(*
触发缩回动作，成功触发返回TRUE，触发失败返回FALSE
*)
METHOD Act_DirectionJog : BOOL
VAR_IN_OUT
	_noteHMI:NoteStruct;
END_VAR
VAR_INPUT
	dir:BOOL;
	vel:DINT;
	len:DINT;
END_VAR
IF enable AND JOGCondition AND NOT busy THEN// AND NOT busy
	// pos:=0;
	// vel:=0;
	jogsetDir:=dir;
	jogsetlen:=len;
	IF (actpos-len>=minPos AND NOT dir) OR (actpos+len<=maxPos AND dir)THEN
		IF jogsetDir THEN
			FuncModule_RS232_ARM.ArmIN(pos:=actpos+len,vel:=setvel,acc:=10);
		ELSE
			FuncModule_RS232_ARM.ArmIN(pos:=actpos-len,vel:=setvel,acc:=10);
		END_IF
		note_IN:=FALSE;
		note_HOME:=FALSE;
		note_JOG:=FALSE;
		IF vel>0 THEN
			jogResetTime:=len/vel;
		END_IF
		jogBusy:=TRUE;
	ELSE
		note_IN:=FALSE;
		note_HOME:=FALSE;
		note_JOG:=TRUE;
		_noteHMI.showFlag:=TRUE;
		_noteHMI.showText:='';
		_noteHMI.showText:=CONCAT(_noteHMI.showText,nameTXT);
		_noteHMI.showText:=CONCAT(_noteHMI.showText,' JOG Condition Not Satisfied!');
	END_IF
	Act_DirectionJog:=TRUE;
ELSE
	Act_DirectionJog:=FALSE;
	note_IN:=FALSE;
	note_HOME:=FALSE;
	note_JOG:=TRUE;
	_noteHMI.showFlag:=TRUE;
	_noteHMI.showText:='';
	_noteHMI.showText:=CONCAT(_noteHMI.showText,nameTXT);
	_noteHMI.showText:=CONCAT(_noteHMI.showText,' JOG Condition Not Satisfied!');
END_IF
END_METHOD

(*
触发缩回动作，成功触发返回TRUE，触发失败返回FALSE
*)
METHOD Act_HOME : BOOL
VAR_IN_OUT
	_noteHMI:NoteStruct;
END_VAR
IF enable AND HOMECondition THEN// AND NOT busy
	// pos:=0;
	// vel:=0;
	Act_HOME:=HOME:=TRUE;
ELSE
	IF gCtrlMode=ControlMode.eManualCtrMode THEN
		note_IN:=FALSE;
		note_HOME:=FALSE;
		note_JOG:=TRUE;
		_noteHMI.showFlag:=TRUE;
		_noteHMI.showText:='';
		_noteHMI.showText:=CONCAT(_noteHMI.showText,nameTXT);
		_noteHMI.showText:=CONCAT(_noteHMI.showText,' HOME Condition Not Satisfied!');
	END_IF
	Act_HOME:=FALSE;
END_IF
END_METHOD

(*
触发缩回动作，成功触发返回TRUE，触发失败返回FALSE
*)
METHOD Act_HOME_Auto : BOOL
IF enable AND HOMECondition THEN// AND NOT busy
	// pos:=0;
	// vel:=0;
	Act_HOME_Auto:=HOME:=TRUE;
ELSE
	Act_HOME_Auto:=FALSE;
END_IF
END_METHOD

(*
触发伸出动作，成功触发返回TRUE，触发失败返回FALSE
*)
METHOD Act_IN : BOOL
VAR_IN_OUT
	_noteHMI:NoteStruct;
END_VAR
IF enable AND INCondition THEN// AND NOT busy
	// pos:=pos;
	// vel:=vel;
	Act_IN:=IN:=TRUE;
ELSE
	IF gCtrlMode=ControlMode.eManualCtrMode THEN
		note_IN:=TRUE;
		note_HOME:=FALSE;
		_noteHMI.showFlag:=TRUE;
		_noteHMI.showText:='';
		_noteHMI.showText:=CONCAT(_noteHMI.showText,nameTXT);
		_noteHMI.showText:=CONCAT(_noteHMI.showText,' IN Condition Not Satisfied!');
	END_IF
	Act_IN:=FALSE;
END_IF
END_METHOD

(*
触发伸出动作，成功触发返回TRUE，触发失败返回FALSE
*)
METHOD Act_IN_Auto : BOOL
IF enable AND INCondition THEN// AND NOT busy
	// pos:=pos;
	// vel:=vel;
	Act_IN_Auto:=IN:=TRUE;
ELSE
	Act_IN_Auto:=FALSE;
END_IF
END_METHOD

(*
触发复位报警动作，成功触发返回TRUE，触发失败返回FALSE
*)
METHOD Act_Reset : BOOL
VAR_INPUT
END_VAR
Act_Reset:=reset:=TRUE;
END_METHOD

(*
触发停止输出动作，成功触发返回TRUE，触发失败返回FALSE
*)
METHOD Act_Stop : BOOL
VAR_INPUT
END_VAR
Act_Stop:=stop:=TRUE;
END_METHOD

ACTION Error_ACT:
CASE errorStep OF
	0:
		error:=FALSE;
		errID:=0;
		errTXT:='';
 (*
	1:
		error:=TRUE;
		errID:=errorID+errorStep;
		errTXT:=CONCAT(STR1:=nameTXT,STR2:=' Extend Error!');
		errWTXT:=WCONCAT(STR1:=TO_WSTRING(nameTXT),STR2:=" 伸出(打开)错误");
	2:
		error:=TRUE;
		errID:=errorID+errorStep;
		errTXT:=CONCAT(STR1:=nameTXT,STR2:=' Retract Error!');
		errWTXT:=WCONCAT(STR1:=TO_WSTRING(nameTXT),STR2:=" 缩回(关闭)错误");
		*)
	1..5:
		error:=TRUE;
		errID:=getErrID(errorStep);
		errTXT:=getErrTXT(errorStep);
		errWTXT:=getErrWTXT(errorStep);
END_CASE
END_ACTION

METHOD Get_Done_HOME : BOOL
VAR_INPUT
END_VAR
Get_Done_HOME:=HOMEdone;
END_METHOD

METHOD Get_Done_IN : BOOL
VAR_INPUT
END_VAR
Get_Done_IN:=INdone;
END_METHOD

METHOD getErrID : UDINT
VAR_INPUT
	errID					:UDINT;//取值范围1~2
END_VAR
VAR
	nErrID					:UDINT;
END_VAR
nErrID:=errorID+errID;

getErrID:=nErrID;
END_METHOD

METHOD getErrTXT : STRING(255)
VAR_INPUT
	errID					:UDINT;//取值范围1~2
END_VAR
VAR
	sErrTXT					:STRING(255);
END_VAR

CASE errID OF
	1:
		sErrTXT:=CONCAT(STR1:=nameTXT,STR2:=' IN Error!');
	2:
		sErrTXT:=CONCAT(STR1:=nameTXT,STR2:=' HOME Error!');
	3:
		sErrTXT:=CONCAT(STR1:=nameTXT,STR2:=' SensorCheck Error!');
	4:
		sErrTXT:=CONCAT(STR1:=nameTXT,STR2:=' Home/IN Time Out Error!');
	5:
		sErrTXT:=CONCAT(STR1:=nameTXT,STR2:=' Communication Error!');
ELSE
	sErrTXT:=CONCAT(STR1:=nameTXT,STR2:='');
END_CASE
getErrTXT:=sErrTXT;
END_METHOD

METHOD getErrWTXT : WSTRING(255)
VAR_INPUT
	errID					:UDINT;//取值范围1~16
END_VAR
VAR
	sErrTXT					:WSTRING(255);
END_VAR

CASE errID OF
	1:
		sErrTXT:=WCONCAT(STR1:=TO_WSTRING(nameTXT),STR2:=" 去工作位错误");
	2:
		sErrTXT:=WCONCAT(STR1:=TO_WSTRING(nameTXT),STR2:=" 回原点错误");
	3:
		sErrTXT:=WCONCAT(STR1:=TO_WSTRING(nameTXT),STR2:=" 传感器检测异常");
	4:
		sErrTXT:=WCONCAT(STR1:=TO_WSTRING(nameTXT),STR2:=" 回原或去目标位超时异常");
	5:
		sErrTXT:=WCONCAT(STR1:=TO_WSTRING(nameTXT),STR2:=" 通讯异常");
ELSE
	sErrTXT:=WCONCAT(STR1:=TO_WSTRING(nameTXT),STR2:="");
END_CASE
getErrWTXT:=sErrTXT;
END_METHOD

ACTION HOME_ACT:
// ARMHOME--HOME 触发
IF HOME AND NOT HOMECondition THEN
	note_HOME:=TRUE;
	note_IN:=FALSE;
	note_JOG:=FALSE;
	NoteHMI.showFlag:=TRUE;
	NoteHMI.showText:='';
	NoteHMI.showText:=CONCAT(NoteHMI.showText,nameTXT);
	NoteHMI.showText:=CONCAT(NoteHMI.showText,' Home Condition Not Satisfied!');
	operatorLog.append(CONCAT(nameTXT,' HOME Not Done'));
END_IF
IF HOME AND enable AND HOMECondition THEN// AND NOT busy
	busy:=TRUE;
	IN:=FALSE;
	INdone:=FALSE;
	HOMEdone:=FALSE;
	INStep:=0;
	HOMEStep:=10;
	note_IN:=FALSE;
	note_HOME:=FALSE;
	note_JOG:=FALSE;
	readAndWriteLock:=TRUE;
	operatorLog.append(CONCAT(nameTXT,' HOME Done'));
	//errorStep:=0;
END_IF
HOME:=FALSE;
// Jog先不考虑，万不得已再使用
// IN ,Home,Jog任意一个Busy；则Recive程序先不动；分别进入程序没发送之类，之后一直采集位置，监控是否到位
CASE HOMEStep OF
0:
	//ready
	
10:
	HOMEErrorDelayTon(IN:=FALSE);
	HOMEDoneDelayTon(IN:=FALSE);
	HOMEStep:=20;
	INRelay:=FALSE;
	HOMERelay:=TRUE;
	FuncModule_RS232_ARM.readSopFlag:=FALSE;
	FuncModule_RS232_ARM.ArmHOME();
15:
	HomedelaycheckTON(IN:=TRUE,PT:=HomedelaycheckTime);
	IF HomedelaycheckTON.Q THEN
		HOMEStep:=20;
		HomedelaycheckTON(IN:=FALSE);
	END_IF
20:
	IF NOT HOMEAprSw OR HOMEAprSw THEN // 读取传感器状态  AND readPos=HomePos
		HOMEStep:=30;
		HOMEErrorDelayTon(IN:=FALSE);
		RETURN;
	END_IF
	HOMEErrorDelayTon(IN:=(NOT HOMEAprSw),PT:=errorDelayTime);// or readPos<>HomePos
	IF HOMEErrorDelayTon.Q THEN
		HOMEStep:=200;
		INdone:=FALSE;
		HOMEdone:=FALSE;
		errorStep:=4;
		HOMEErrorDelayTon(IN:=FALSE);
	END_IF
	
30:
	HOMEStep:=100;
	readAndWriteLock:=FALSE;
100:
	HOMEErrorDelayTon(IN:=(NOT HOMEAprSw),PT:=errorDelayTime);// rec pos=setpos or SW HOME Sensor
	IF HOMEErrorDelayTon.Q THEN
		//done:=FALSE;
		INdone:=FALSE;
		HOMEdone:=FALSE;
		errorStep:=2;
		HOMEStep:=200;
		RETURN;
	END_IF
	IF enableHOMEAprSw THEN
		HOMEDoneDelayTon(IN:=HOMEAprSw AND FuncModule_RS232_ARM.readSopFlag,PT:=doneDelayTimeShortHOME);
	ELSE
		HOMEDoneDelayTon(IN:=NOT enableHOMEAprSw,PT:=doneDelayTimeLongHOME);
	END_IF
	
	IF HOMEDoneDelayTon.Q THEN
		IF HOMEAprSw THEN
			busy:=FALSE;
			//done:=TRUE;
			INdone:=FALSE;
			HOMEdone:=TRUE;
			errorStep:=0;
			HOMEStep:=150;
		ELSE
			busy:=FALSE;
			//done:=TRUE;
			INdone:=FALSE;
			HOMEdone:=FALSE;
			errorStep:=2;
			HOMEStep:=200;
		END_IF
	END_IF
150:
	readAndWriteLock:=FALSE;
	HOMEStep:=0;
200:
	readAndWriteLock:=FALSE;
	HOMEStep:=0;
END_CASE
END_ACTION

ACTION IN_ACT:
//气缸伸出--IN 触发
IF IN AND NOT INCondition THEN
	note_IN:=TRUE;
	note_HOME:=FALSE;
	note_JOG:=FALSE;
	NoteHMI.showFlag:=TRUE;
	NoteHMI.showText:='';
	NoteHMI.showText:=CONCAT(NoteHMI.showText,nameTXT);
	NoteHMI.showText:=CONCAT(NoteHMI.showText,' IN Condition Not Satisfied!');
	operatorLog.append(CONCAT(nameTXT,' In Not Done'));
END_IF
IF IN AND enable AND INCondition THEN// AND NOT busy
	busy:=TRUE;
	HOME:=FALSE;
	INdone:=FALSE;
	HOMEdone:=FALSE;
	INStep:=10;
	HOMEStep:=0;
	note_IN:=FALSE;
	note_HOME:=FALSE;
	note_JOG:=FALSE;
	readAndWriteLock:=TRUE;
	operatorLog.append(CONCAT(CONCAT(nameTXT,' IN'),DINT_TO_STRING(setvel)));
	//errorStep:=0;
END_IF
IN:=FALSE;
// Jog先不考虑，万不得已再使用
// IN ,Home,Jog任意一个Busy；则Recive程序先不动；分别进入程序没发送之类，之后一直采集位置，监控是否到位
CASE INStep OF
0:
	//ready
	
10:
	INErrorDelayTon(IN:=FALSE);
	INDoneDelayTon(IN:=FALSE);
	IndelaycheckTON(IN:=FALSE);
	INStep:=15;
	INRelay:=TRUE;
	FuncModule_RS232_ARM.readSopFlag:=FALSE;
	FuncModule_RS232_ARM.ArmIN(pos:=setpos,vel:=setvel,acc:=10);
	// send:vel
	HOMERelay:=FALSE;
15:
	IndelaycheckTON(IN:=TRUE,PT:=IndelaycheckTime);
	IF IndelaycheckTON.Q THEN
		INStep:=20;
		IndelaycheckTON(IN:=FALSE);
	END_IF
20:
	IF NOT HOMEAprSw (*AND readPos=InPos*) THEN // 读取数据，判断接收的数据是否是设定的Vel；
		INStep:=30;
		INErrorDelayTon(IN:=FALSE);
		RETURN;
	ELSE
		INStep:=15;
	END_IF
	INErrorDelayTon(IN:=(HOMEAprSw (*OR readPos<>InPos*) ),PT:=errorDelayTime);
	IF INErrorDelayTon.Q THEN
		INStep:=200;
		INdone:=FALSE;
		HOMEdone:=FALSE;
		errorStep:=4;
		INErrorDelayTon(IN:=FALSE);
	END_IF
	
30:
	// send:pos
	INStep:=100;
	readAndWriteLock:=FALSE;
	
100:
	INErrorDelayTon(IN:=(HOMEAprSw OR NOT FuncModule_RS232_ARM.readSopFlag),PT:=errorDelayTime);// rec pos=setpos or SW IN Sensor
	IF INErrorDelayTon.Q THEN
		//done:=FALSE;
		INdone:=FALSE;
		HOMEdone:=FALSE;
		errorStep:=1;
		INStep:=200;
		RETURN;
	END_IF
	IF enableINAprSw THEN// Run则通过指令知道设备在什么地方
		INDoneDelayTon(IN:=NOT HOMEAprSw AND FuncModule_RS232_ARM.readSopFlag,PT:=doneDelayTimeShortIN);// rec pos=setpos
	ELSE
		INDoneDelayTon(IN:=NOT enableINAprSw,PT:=doneDelayTimeLongIN);
	END_IF
	
	IF INDoneDelayTon.Q THEN
		IF NOT HOMEAprSw THEN
			busy:=FALSE;
			//done:=TRUE;
			INdone:=TRUE;
			HOMEdone:=FALSE;
			errorStep:=0;
			INStep:=150;
		ELSE
			busy:=FALSE;
			//done:=TRUE;
			INdone:=FALSE;
			HOMEdone:=FALSE;
			errorStep:=1;
			INStep:=200;
		END_IF
	END_IF
150:
	readAndWriteLock:=FALSE;
	INStep:=0;
200:
	readAndWriteLock:=FALSE;
	INStep:=0;
END_CASE
END_ACTION

ACTION Init_ACT:
done:=(INdone OR HOMEdone);
InitHMI_ACT();
manualCtrl_ACT();

IF NOT FuncModule_RS232_ARM.serialConnected AND firstPowerTON.Q THEN
	errorStep:=5;
END_IF
noteTON_P(IN:=note_IN,PT:=T#0.1S);
noteRTrig_P(CLK:=noteTON_P.Q);
IF noteRTrig_P.Q THEN
//	gLog_Note.append_EX(noteWTXT_Ext);
END_IF
noteTON_N(IN:=note_HOME,PT:=T#0.1S);
noteRTrig_N(CLK:=noteTON_N.Q);
IF noteRTrig_N.Q THEN
//	gLog_Note.append_EX(noteWTXT_Ret);
END_IF

jogResetTON(in:=jogBusy,PT:=DINT_TO_TIME(jogResetTime*1000));
IF jogResetTON.Q THEN
	jogBusy:=FALSE;
END_IF
END_ACTION

ACTION InitHMI_ACT:
HMIItf.INAprSw:=INAprSw;
HMIItf.HOMEAprSw:=HOMEAprSw;
HMIItf.enableIN:=enableINAprSw;
HMIItf.enableHOME:=enableHOMEAprSw;
HMIItf.HMIEnable:=hmiEN;
HMIItf.enable:=enable;
HMIItf.done:=done;
HMIItf.busy:=busy;
HMIItf.error:=error;
HMIItf.errID:=UDINT_TO_DINT(errID);
HMIItf.errTXT:=errTXT;
HMIItf.INRelay:=INRelay;
HMIItf.HOMERelay:=HOMERelay;
HMIItf.power:=power;
HMIItf.nameTXT:=nameTXT;
HMIItf.extenderror:=error AND errorID=1;
HMIItf.retracterror:=error AND errorID=2;
HMIItf.INcondition:=INCondition;
HMIItf.HOMEcondition:=HOMECondition;
END_ACTION

ACTION ManualCtrl_ACT:
//HMI手动控制
//IF ctrlMode=eManualCtrMode THEN
IF hmiEN THEN
	INTrigRAlc(CLK:=HMIItf.INAndHOME);
	IF INTrigRAlc.Q THEN// AND NOT busy
		IF INRelay THEN//如果伸出继电器或伸出传感器亮，则认为已经伸出过
			HOME:=TRUE;
		END_IF
		IF HOMERelay THEN
			IN:=TRUE;
		END_IF
		IF NOT INRelay AND NOT HOMERelay THEN
			IF INAprSw THEN
				HOME:=TRUE;
			END_IF
			IF HOMEAprSw THEN
				IN:=TRUE;
			END_IF
		END_IF
	END_IF
	INTrigR1(CLK:=HMIItf.IN);
	IF INTrigR1.Q THEN// AND NOT busy
		WarmHMI.showText:='';
		WarmHMI.showFlag:=TRUE;
		WarmHMI.showText:=CONCAT(WarmHMI.showText,'Are you sure you want the ');
		WarmHMI.showText:=CONCAT(WarmHMI.showText,nameTXT);
		WarmHMI.showText:=CONCAT(WarmHMI.showText,' to INChamber?');
	END_IF
	IF WarmHMI.bOK AND NOT WarmHMI.showFlag AND FIND(WarmHMI.showText,nameTXT)>0 AND FIND(WarmHMI.showText,'INChamber')>0 THEN
		IN:=TRUE;
		WarmHMI.bOK:=FALSE;
		WarmHMI.showText:='';
	END_IF
	IF WarmHMI.bNO AND NOT WarmHMI.showFlag AND FIND(WarmHMI.showText,nameTXT)>0 AND FIND(WarmHMI.showText,'INChamber')>0 THEN
		WarmHMI.bNO:=FALSE;
		WarmHMI.showText:='';
	END_IF
	
	HOMETrigR1(CLK:=HMIItf.HOME);
	IF HOMETrigR1.Q THEN// AND NOT busy
		WarmHMI.showText:='';
		WarmHMI.showFlag:=TRUE;
		WarmHMI.showText:=CONCAT(WarmHMI.showText,'Are you sure you want to the ');
		WarmHMI.showText:=CONCAT(WarmHMI.showText,nameTXT);
		WarmHMI.showText:=CONCAT(WarmHMI.showText,' to Homing?');
	END_IF
	IF WarmHMI.bOK AND NOT WarmHMI.showFlag AND FIND(WarmHMI.showText,nameTXT)>0 AND FIND(WarmHMI.showText,'Homing')>0 THEN
		HOME:=TRUE;
		WarmHMI.bOK:=FALSE;
		WarmHMI.showText:='';
	END_IF
	IF WarmHMI.bNO AND NOT WarmHMI.showFlag AND FIND(WarmHMI.showText,nameTXT)>0 AND FIND(WarmHMI.showText,'Homing')>0 THEN
		WarmHMI.bNO:=FALSE;
		WarmHMI.showText:='';
	END_IF
	
	resetTrigR1(CLK:=HMIItf.reset);
	IF resetTrigR1.Q THEN// AND NOT busy
		reset:=TRUE;
	END_IF
	
	stopTrigR1(CLK:=HMIItf.stop);
	IF stopTrigR1.Q THEN// AND NOT busy
		stop:=TRUE;
	END_IF
	
	powerTrigR1(CLK:=HMIItf.power);
	IF powerTrigR1.Q THEN// AND NOT busy
		IF power THEN
			power:=FALSE;
		ELSE
			power:=TRUE;
		END_IF
	END_IF
END_IF
END_ACTION

ACTION Read_ACT:
//气缸收回--read 触发
firstPowerTON(IN:=firstPower,PT:=T#5S);
IF NOT readAndWriteLock AND NOT readbusy AND readStep=0 AND readCondition THEN// AND NOT busy
	readdone:=FALSE;
	readStep:=10;
	readbusy:=TRUE;
	readerror:=FALSE;
END_IF
CASE readStep OF
0:
	//ready
	readTon1(IN:=FALSE);
	readTon2(IN:=FALSE);
10:// State
	IF readAndWriteLock THEN
		readStep:=5000;
	ELSE
		FuncModule_RS232_ARM.readPosFlag:=FALSE;
		FuncModule_RS232_ARM.GetPos();
		readStep:=readStep+10;
	END_IF
20:
	IF readAndWriteLock THEN
		readStep:=5000;
	ELSE
		IF FuncModule_RS232_ARM.readPosFlag THEN
			FuncModule_RS232_ARM.readPosFlag:=FALSE;
			// 数据处理
			actpos:=FuncModule_RS232_ARM.POS;
			readTon1(IN:=FALSE);
			readStep:=25;
			RETURN;
		END_IF
		readTon1(IN:=TRUE,PT:=T#500MS);// 超时
		IF readTon1.Q THEN
			readStep:=6000;
			readTon1(IN:=FALSE);
			readTon2(IN:=FALSE);
			RETURN;
		END_IF
		;
	END_IF
25:
	t1(IN:=TRUE,PT:=T#0.5S);
	IF t1.Q THEN
		readStep:=5000;
		t1(IN:=FALSE);
	END_IF
100:// Internal RTD1
	IF readAndWriteLock THEN
		readStep:=5000;
	ELSE
		FuncModule_RS232_ARM.readStateFlag:=FALSE;
		FuncModule_RS232_ARM.GetState();
		readStep:=readStep+10;
	END_IF	
110:
	IF readAndWriteLock THEN
		readStep:=5000;
	ELSE
		IF FuncModule_RS232_ARM.readStateFlag THEN
			FuncModule_RS232_ARM.readStateFlag:=FALSE;
			// 数据处理
			readTon1(IN:=FALSE);
			readStep:=5000;
			RETURN;
		END_IF
		readTon1(IN:=TRUE,PT:=T#500MS);// 超时
		IF readTon1.Q THEN
			readStep:=6000;
			readTon1(IN:=FALSE);
			readTon2(IN:=FALSE);
			RETURN;
		END_IF
		;
	END_IF
	
5000:
	readbusy:=FALSE;
	readdone:=TRUE;
	readStep:=0;
	readerror:=FALSE;
6000:
	readbusy:=FALSE;
	readdone:=TRUE;
	readStep:=0;
	readerror:=TRUE;
END_CASE
END_ACTION

ACTION RealMonitor_ACT:
notBusyMonitorDelayTon(IN:=NOT busy,PT:=notBusyMonitorDelayTime);
IF real_TimeMonitor THEN
	IF notBusyMonitorDelayTon.Q THEN
		//伸出实时检测
//		IF (enableINAprSw AND NOT INAprSw) AND INRelay THEN
//			errorStep:=1;
//		END_IF
	
//		//缩回实时检测	
//		IF (enableINAprSw AND NOT HOMEAprSw) AND HOMERelay  THEN
//			errorStep:=2;
//		END_IF
	END_IF
END_IF
END_ACTION

ACTION Reset_ACT:
IF reset THEN
	IF NOT power THEN
		INRelay:=FALSE;
		HOMERelay:=FALSE;
	END_IF
	busy:=FALSE;
	//done:=FALSE;
	//extdone:=FALSE;
	//retdone:=FALSE;
	errorStep:=0;
	note_IN:=FALSE;
	note_HOME:=FALSE;
	note_JOG:=FALSE;
	reset:=FALSE;
END_IF

IF stop THEN
	stop:=FALSE;
	INRelay:=FALSE;
	HOMERelay:=FALSE;
	note_IN:=FALSE;
	note_HOME:=FALSE;
	note_JOG:=FALSE;
	busy:=FALSE;
	INStep:=0;
	HOMEStep:=0;
	FuncModule_RS232_ARM.ArmStop();
	//无自锁检测说法，直接停
//	extStep:=0;
//	retStep:=0;
END_IF
END_ACTION

ACTION VersionLog:
(*
版本: V1.0.0.0
说明:
	1. 首个版本
	2. 含普通气缸\真空吸类型的控制
	3. 可配置是否有到位信号, 以及到位稳定时间
(--------------------------------------------------)
新版本: V1.0.1.0
更新时间: 2019/11/20 19:00
更新说明:
	1. 优化编写方式
	2. 修改错误编码起始位，现改为从1开始
(--------------------------------------------------)
新版本: V1.0.1.1
更新时间: 2020/03/23 23:00
更新说明:
	1. 优化报错方式
	2. 增加伸出、缩回、复位和停止触发函数
(--------------------------------------------------)
新版本: V1.0.1.2
更新时间: 2020/04/22 09:50
更新说明:
	1. 增加中文报警输出
(--------------------------------------------------)
新版本: V1.0.1.3
更新时间: 2020/09/16
更新说明:
	1. 开放错误ID、错误文本信息获取接口
(--------------------------------------------------)
新版本: V1.0.1.4
更新时间: 2020/10/06
更新说明:
	1. 移除控制模式变量，增加HMI启用条件
	2. 增加外部获取伸出缩回完成信号接口函数
(--------------------------------------------------)
新版本: V1.0.1.5
更新时间: 2020/10/14
更新说明:
	1. 优化代码
(--------------------------------------------------)
*)
END_ACTION

END_FUNCTION_BLOCK

// ---- POUs/BaseModule/Communication/FuncModule_RS232_ARM.TcPOU
PROGRAM FuncModule_RS232_ARM
VAR_INPUT
	serialExcute				:BOOL;// RS232开始一次参数读取
	serialSlaveID				:UINT;// 232从站节点号
	sendstr						:STRING;
	prefix						:STRING:='';// 字符串头
	suffix						:STRING:= '';// 字符串尾
	timeout						:TIME:=T#200MS;// 超时时间
	goPosLoad					:LREAL;
	goPosPhase					:LREAL;
	setPresetExt				:BOOL;
	readPosFlag					:BOOL;
	readStateFlag				:BOOL;
	readSopFlag					:BOOL;// 停止标志位
END_VAR
VAR_OUTPUT
	serialBusy						:BOOL;
	setPresetBusy					:BOOL;
	serialDone						:BOOL;
	setPresetDone						:BOOL;
	serialError						:BOOL;
	setPresetError						:BOOL;
	serialConnected					:BOOL;
	POS							:INT;// 
	oldPOS							:int;// 
	phase							:REAL;// Phase电容
	rec_ManulOrAuto					:BOOL;// Manul OR Auto
	rec_MAStr						:STRING:='Auto';
	loadRunErr						:BOOL;
	phashRunErr						:BOOL;
END_VAR
VAR
	//Byte方式
	send1:							SendData;
	receive1:						ReceiveString;
 
	Timer1:							TON;
	TimerSetPreset:							TON;
	t1:								TON;
	ITemp:INT;
	arr_SendData:					STRING;(*READ*)//发送数据
	arr_RcvDataString:				STRING;// 接收数据
	arr_RcvDataStringTemp:				STRING;// 接收数据
	arr_RcvDataStringClear:			STRING;// 清除接收数据
	RcvDataFlag:			BOOL;// 接收数据标志位
	serialStep						:UINT;				//处理步数
	serialErrorID					:UINT;
	setPresetStep					:UINT;				//处理步数
	serialTimeOut:BOOL;//接收数据超时
	serialRecError:BOOL;//接收数据错误
	reciveFtrig:F_TRIG;
	recTon:TON;
	againSendS3:TON;
	//字符串方式
	(*send1:							SendString;
	receive1:						ReceiveString;
	
	Timer1:							TON;
	
	_sendString:					STRING:='4567';
	_receive1string:				STRING;
	_recvLast:						STRING;				//保存上一个周期接收的字符*)

	
	decimalvalue:INT;
	decimalvalueP:INT;
	hexString:STRING(8);
	hexStringP:STRING(8);
	i:INT;
	hexChars:ARRAY [0..15] OF STRING[1]:=['0','1','2','3','4','5','6','7','8','9','A','B','C','D','E','F'];
	index:INT;
	findposstart	:INT;
	findposend		:INT;
	find_pos		:INT;
	recStrTemp		:STRING(255);
END_VAR

(*
 *功能块的作用，把 TxBuffer 缓存区的数据经过 Process Data 的 ComOut 发送出去，
 *而把 ComIn 中的数据接收到 RxBuffer。引用这个功能块的程序执行周期越短，
 *数据交换的效率就越高，所以这段程序应该放在快速任务中作为 Backgroud 代码无条件执行。
*)
IF receive1.Error <> COMERROR_NOERROR THEN
	serialRecError:=TRUE;
END_IF
receive1(
	Prefix:= prefix, 
	Suffix:= suffix, 
	Timeout:=timeout , 
	Reset:= , 
	StringReceived=> , 
	Busy=> , 
	Error=> , 
	RxTimeout=> , 
	ReceivedString:= arr_RcvDataStringTemp, 
	RXbuffer:=gRxBuffer_ARM );

//testReal:=BYTE_TO_REAL(arr_RcvData_Temp);
//数据接收处理
reciveFtrig(CLK:=receive1.busy);
IF reciveFtrig.Q THEN
	arr_RcvDataString:=arr_RcvDataStringTemp;
	arr_RcvDataStringTemp:=arr_RcvDataStringClear;
	RcvDataFlag:=TRUE;
	serialConnected:=TRUE;
END_IF
recTon(IN:=RcvDataFlag, PT:=T#20MS);
IF recTon.Q THEN
	RcvDataFlag:=FALSE;
END_IF
againSendS3(IN:=NOT RcvDataFlag,PT:=T#5S);
IF againSendS3.Q THEN
	serialConnected:=FALSE;
	againSendS3(IN:=FALSE);
END_IF

ACT_Send();

ACT_RcvProcess();

ACTION ACT_RcvProcess:
find_pos:=0;
findposend:=0;
findposstart:=0;

IF MID(arr_RcvDataString,3,1)='?96' THEN
	recStrTemp:=DELETE(arr_RcvDataString,5,1);
	IF MID(recStrTemp,5,1)='Px.1='  THEN
		readPosFlag:=TRUE;
		IF  MID(recStrTemp,1,6)='-' THEN
			POS:=oldPOS+STRING_TO_INT(MID(recStrTemp,LEN(recStrTemp)-7,6));
		ELSE
			POS:=STRING_TO_INT(MID(recStrTemp,LEN(recStrTemp)-7,6));
			oldPOS:=POS;
		END_IF
	END_IF
END_IF

IF FIND(arr_RcvDataString,'Ux.1=8')>0 THEN
	readSopFlag:=TRUE;
END_IF
END_ACTION

ACTION ACT_Send:

CASE serialStep OF
	0:
	IF serialExcute THEN
		serialExcute:=FALSE;
		IF NOT serialBusy THEN
			serialStep:=90;
			serialBusy:=TRUE;
			serialDone:=FALSE;
			serialError:=FALSE;
			serialTimeOut:=FALSE;
			serialRecError:=FALSE;
		END_IF
	END_IF
	Timer1(IN:= FALSE);
	;
	90:
		arr_SendData:=sendstr;
		serialStep:=100;
	100:
		send1(
			pSendData:= ADR(arr_SendData), 
			Length:= INT_TO_UDINT(LEN(arr_SendData)), 
			Busy=> , 
			Error=> , 
			TXbuffer:= gTxBuffer_ARM);
		serialStep:=serialStep+10;
	110:
		Timer1(IN:= NOT timer1.q, PT:=T#10MS);
		IF Timer1.Q THEN
			serialStep:=serialStep+10;
			Timer1(IN:= FALSE);
		END_IF
	120:
		Timer1(IN:= NOT timer1.q, PT:=T#500MS);
		IF Timer1.Q THEN
			serialStep:=6000;
			Timer1(IN:= FALSE);
			serialTimeOut:=TRUE;
			RETURN;
		END_IF
		IF NOT send1.busy  THEN
			Timer1(IN:= FALSE);
			serialTimeOut:=FALSE;
			serialStep:=200;
		END_IF
		IF send1.Error <> COMERROR_NOERROR THEN
			serialRecError:=TRUE;
		END_IF
	200://数据处理
		serialStep:=serialStep+10;
	210:
		Timer1(IN:= NOT timer1.q, PT:=T#10MS);
		IF Timer1.Q THEN
			serialStep:=serialStep+10;
			Timer1(IN:= FALSE);
		END_IF
	220:
		//数据转换
		Timer1(IN:= FALSE);
		serialStep:=1000;
	
	1000:
		Timer1(IN:= NOT timer1.q, PT:=T#50MS);
		IF Timer1.Q THEN
			serialStep:=5000;
			Timer1(IN:= FALSE);
			// sendstr:='';
			serialTimeOut:=FALSE;
		END_IF
	;
	5000://done
		serialBusy:=FALSE;
		serialDone:=TRUE;
		serialError:=FALSE;
		serialStep:=0;
	;
	6000://error
		serialBusy:=FALSE;
		serialDone:=FALSE;
		serialError:=TRUE;
		serialStep:=0;
	;
	
END_CASE
END_ACTION

METHOD ArmHOME : BOOL
VAR_INPUT
END_VAR
sendstr:='';
sendstr:='|$R';
serialExcute:=TRUE;
END_METHOD

METHOD ArmIN : BOOL
VAR_INPUT
	pos:DINT;
	vel:DINT;
	acc:DINT;
END_VAR
VAR
	str:STRING;
END_VAR
str:='';
str:=CONCAT(str,'P=');
str:=CONCAT(str,DINT_TO_STRING(pos));
str:=CONCAT(str,',S=');
str:=CONCAT(str,DINT_TO_STRING(vel));
str:=CONCAT(str,',A=');
str:=CONCAT(str,DINT_TO_STRING(acc));
str:=CONCAT(str,',^$R');
sendstr:='';
sendstr:=str;
serialExcute:=TRUE;
END_METHOD

METHOD ArmStop : BOOL
VAR_INPUT
END_VAR
VAR
	diraction:STRING:='+';
	str:STRING;
END_VAR
str:='';
str:=CONCAT(str,']$R');
sendstr:='';
sendstr:=str;
serialExcute:=TRUE;
END_METHOD

METHOD CalASII_Str : STRING
VAR_INPUT
	date1:UINT;
END_VAR
IF date1=10 THEN
	CalASII_Str:='A';
END_IF
IF date1=11 THEN
	CalASII_Str:='B';
END_IF
IF date1=12 THEN
	CalASII_Str:='C';
END_IF
IF date1=13 THEN
	CalASII_Str:='D';
END_IF
IF date1=14 THEN
	CalASII_Str:='E';
END_IF
IF date1=15 THEN
	CalASII_Str:='F';
END_IF
IF date1<10 THEN
	CalASII_Str:=UINT_TO_STRING(date1);
END_IF
IF date1>15 THEN
	CalASII_Str:=UINT_TO_STRING(date1);
END_IF
END_METHOD

METHOD CalMeth : INT
VAR_INPUT
	byteIn:BYTE;
END_VAR
VAR_OUTPUT
	outInt:INT;
END_VAR
IF byteIn>=48 AND byteIn<=57 THEN
	outInt:=byteIn-48;
ELSE
	outInt:=byteIn-65+10;
END_IF
CalMeth:=outInt;
END_METHOD

METHOD GetPos : BOOL
VAR_INPUT
END_VAR
VAR
	str:STRING;
END_VAR
str:='?96$R';
sendstr:='';
sendstr:=str;
serialExcute:=TRUE;
END_METHOD

METHOD GetState : BOOL
VAR_INPUT
END_VAR
VAR
	str:STRING;
END_VAR
str:='GetState^';
sendstr:='';
sendstr:=str;
serialExcute:=TRUE;
END_METHOD

METHOD IncN : BOOL
VAR_INPUT
	dis:DINT;
	vel:DINT;
	acc:DINT;
END_VAR
VAR
	diraction:STRING:='+';
	str:STRING;
END_VAR
str:='';
str:=CONCAT(str,'P:');
str:=CONCAT(str,DINT_TO_STRING(dis));
str:=CONCAT(str,',S:');
str:=CONCAT(str,DINT_TO_STRING(vel));
str:=CONCAT(str,',A:');
str:=CONCAT(str,DINT_TO_STRING(acc));
str:=CONCAT(str,',D:');
str:=CONCAT(str,diraction);
str:=CONCAT(str,',^$R');
sendstr:='';
sendstr:=str;
serialExcute:=TRUE;
END_METHOD

METHOD IncP : BOOL
VAR_INPUT
	dis:DINT;
	vel:DINT;
	acc:DINT;
END_VAR
VAR
	diraction:STRING:='+';
	str:STRING;
END_VAR
str:='';
str:=CONCAT(str,'P:');
str:=CONCAT(str,DINT_TO_STRING(dis));
str:=CONCAT(str,',S:');
str:=CONCAT(str,DINT_TO_STRING(vel));
str:=CONCAT(str,',A:');
str:=CONCAT(str,DINT_TO_STRING(acc));
str:=CONCAT(str,',D:');
str:=CONCAT(str,diraction);
str:=CONCAT(str,',^$R');
sendstr:='';
sendstr:=str;
serialExcute:=TRUE;
END_METHOD

END_PROGRAM

// ---- POUs/BaseModule/ActionModule/RFModule_Source/RFModule_Source.TcPOU
(*
--报错编号0: 无报错
--报错编号1: openend Error
--报错编号2: close Error
*)
FUNCTION_BLOCK RFModule_Source
VAR_IN_OUT
	WarmHMI					:WARMStruct;
	NoteHMI					:NoteStruct;
	operatorLog				:printLogModule_EX;
END_VAR
VAR_INPUT
	HMIItf						:RFHMIStruts;// 每个RF对象都关联了一个HMI
	RFTYPE						:RFType:=RFType_Default;// 设置RF的类型
	real_TimeMonitor			:BOOL:=TRUE;//实时状态检测
	co_control					:BOOL;// 共同计时
	open						:BOOL:=FALSE;//启动触发信号
	openCondition				:BOOL:=TRUE;//启动条件
	close						:BOOL:=FALSE;//停止触发信号
	closeCondition				:BOOL:=TRUE;//停止条件
	reset						:BOOL:=FALSE;//复位信号
	readCondition				:BOOL:=TRUE;//读取条件
	stop						:BOOL:=FALSE;//停止信号
	power						:BOOL:=TRUE;// RF动作后是否关闭继电器得电状态, TRUE--保持得电,FALSE--断开得电
	enable						:BOOL:=TRUE;// RF禁用条件
	//ctrlMode					:ControlMode:=ControlMode.eManualCtrMode;//eManualCtrMode or eAutoCtrMode
	hmiEN						:BOOL:=TRUE;//HMI 启用条件
	serialExcute				:BOOL;// RS485、232开始一次参数读取
	
	errorDelayTime				:TIME:=T#10S;//分子泵感应器感应超时
	
	ACCMaxtime					:TIME:=T#20S;// RF加速最大时间 启动过程
	DCCMaxtime					:TIME:=T#20S;// RF减速最大时间 停止过程
	
	doneDelayTimeShortopenend	:TIME:=T#100MS;//  RF启动感应到位延时_伸出
	doneDelayTimeShortcloseract	:TIME:=T#50MS;//  RF感应到位延时_收回
	doneDelayTimeLongopenend	:TIME:=T#500MS;//  RF感应到位延时_伸出
	doneDelayTimeLongcloseract	:TIME:=T#50MS;// RF感应到位延时_收回
	errorID						:UDINT:=0;// RF错误报警分配的起始ID
	nameTXT						:STRING(255):='';// RF名字
	
	AlmAprSw					:BOOL:=FALSE;// RF报警感应器信号,需要链接到实际的IO点
	ErrorAprSw					:BOOL:=FALSE;// RF报错感应器信号,需要链接到实际的IO点
	enableOpenAprSw				:BOOL:=TRUE;// 启用启动感应器,针对只有一个传感器的 RF
	enableCloseAprSw			:BOOL:=TRUE;// 启用停止感应器,针对只有一个传感器的 RF
	runTime						: LINT;// 运行时间
	mainPower					:BOOL;// RF主电源
	temperature					:REAL;// RF温度
	current						:REAL;// RF电流
	vol							:REAL;// RF电压
	serialSlaveID				:UINT;// RF ID
	serialError					:BOOL;// RF通讯错误
	setpower					:UDINT;// 设定功率	
	settime						:UDINT;// 设定时间
	noteWTXT_open				:WSTRING(255):="";// RF打开动作NoteTXT 中文
	noteWTXT_close				:WSTRING(255):="";// RF关闭动作NoteTXT 中文
	controlMode					:INT:=0;// 0 手动，1 Analog，2 RS232
	outputMode					:INT:=0;// 0 continuous，1 pulse
	outputState					:INT:=0;// 0 Stop,1 Start
	alarmState					:INT:=0;// 0 No Error,1 Error
	setpowerRead				:UDINT:=0;// 读取设置的功率值
	forwardpower				:UDINT;// 实际功率	
	reflectedpower				:UDINT;// 反馈功率
	maxpower					:UDINT;// 设置的最大功率值
END_VAR
VAR_OUTPUT
	note_open				:BOOL;// 开条件不满足提示
	note_close				:BOOL;// 关条件不满足提示
	openRelay				:BOOL:=FALSE;// RF启动执行继电器,需要链接到实际的IO点
	closeRelay				:BOOL:=FALSE;// RF停止执行继电器,需要链接到实际的IO点
	resetRelay				:BOOL:=FALSE;// RF复位执行继电器,需要链接到实际的IO点	
	rematime				:UDINT;// 剩余时间
	busy					:BOOL;// RFusy状态
	openbusy				:BOOL;// RF开动作Busy状态
	closebusy				:BOOL;// RF关动作Busy状态
	readbusy				:BOOL;// RF循环读取Busy状态
	done					:BOOL;// RF动作Done状态
	readdone					:BOOL;// RF动作Done状态
	opendone				:BOOL;// RF动作伸出完成
	closedone				:BOOL;// RF动作收回完成
	setpointdone			:BOOL;
	readerror			    :BOOL;// RF动作error状态
	error					:BOOL;// RF动作error状态
	errID					:UDINT;// RF动作errID
	errTXT					:STRING(255):='';// RF动作errTXT
	errWTXT					:WSTRING(255):="";// RF动作errTXT 中文
END_VAR
	
VAR	
	readAndWriteLock:BOOL;
	runTON					: TON;
	openErrorDelayTon		:Ton;
	openDoneDelayTon		:Ton;
	closeErrorDelayTon		:Ton;
	closeDoneDelayTon		:Ton;
	
	extendTrigRAlc			:R_Trig;//上升沿触发
	runTimeClearR			:R_Trig;//上升沿触发
	
	openendTrigRAlc			:R_Trig;//上升沿触发
	
	singleControltempR			:R_Trig;//上升沿触发
	singleControlR			:R_Trig;//上升沿触发
	singleControlF			:F_Trig;//上升沿触发
	
	openendTrigR1			:R_Trig;//上升沿触发
	openendTrigR1_Aiko		:R_Trig;//上升沿触发
	closeractTrigR1			:R_Trig;//上升沿触发
	resetTrigR1				:R_Trig;//上升沿触发
	stopTrigR1				:R_Trig;//上升沿触发
	powerTrigR1				:R_Trig;//上升沿触发
	
	openStep				:UINT:=0;
	closeStep				:UINT:=0;
	errorStep				:UINT:=0;
	readStep				:UINT:=0;
	
	resetRelayTON			:TON;
	resetRelayTONTime		:TIME:=T#2S;
	
	writeStep				:UINT:=0;
	writeMaxStep			:UINT:=0;
	
	notBusyMonitorDelayTon:TON;//动作不切换时，延迟检测
	notBusyMonitorDelayTime:TIME:=T#2S;//动作不切换延迟检测时间
	firstPower			    :BOOL:=TRUE;//首次上电标志位
	firstPowerTON			:TON;
	
	AccFTrig:F_TRIG;//检测加速信号下降延
	NormalRTrig:R_TRIG;//匀速上升沿
	DccFTrig:F_TRIG;// 检测减速信号下降延
	noteTON_P:tON;            // 操作提示标志位延时继电器
	noteTON_N:tON;            // 操作提示标志位延时继电器
	noteRTrig_P:R_TRIG;          // 操作提示
	noteRTrig_N:R_TRIG;          // 操作提示
	powerTon:TON;
	readTon1:TON;
	readTon2:TON;
	readTon3:TON;
	t1:TON;
	t2:TON;
	writeTON:TON;
	writeMaxTON:TON;
	readTON:TON;
	readErrorTimes:UINT:=0;
END_VAR

Init_ACT();
Error_ACT();
Open_ACT();
Close_ACT();
Reset_ACT();
Error_ACT();
Read_ACT();
WritePower_ACT();
WriteMaxPower_ACT();

(*
触发缩回动作，成功触发返回TRUE，触发失败返回FALSE
*)
METHOD Act_Close : BOOL
VAR_INPUT
END_VAR
IF enable AND closeCondition THEN// AND NOT busy
	Act_Close:=close:=TRUE;
ELSE
	Act_Close:=FALSE;
END_IF
END_METHOD

(*
触发伸出动作，成功触发返回TRUE，触发失败返回FALSE
*)
METHOD Act_Open : BOOL
VAR_INPUT
END_VAR
IF enable AND openCondition THEN// AND NOT busy
	Act_Open:=open:=TRUE;
ELSE
	Act_Open:=FALSE;
END_IF
END_METHOD

(*
触发复位报警动作，成功触发返回TRUE，触发失败返回FALSE
*)
METHOD Act_Reset : BOOL
VAR_INPUT
END_VAR
Act_Reset:=reset:=TRUE;
END_METHOD

(*
触发发送动作，成功触发返回TRUE，触发失败返回FALSE
*)
METHOD Act_SerialSend : BOOL
VAR_INPUT
END_VAR
IF TRUE THEN
	Act_SerialSend:=serialExcute:=TRUE;
ELSE
	Act_SerialSend:=FALSE;
END_IF
END_METHOD

METHOD Act_SetPoint : BOOL
VAR_INPUT
	setpoint:UDINT;
	_settime:UDINT;
	con_ctr:BOOL;
END_VAR
VAR_OUTPUT
	outTime:UDINT;
END_VAR
setpower:=HMIItf.setpower:=setpoint;
settime:=HMIItf.settime:=outTime:=_settime;
co_control:=con_ctr;
Act_Open();
END_METHOD

(*
触发停止输出动作，成功触发返回TRUE，触发失败返回FALSE
*)
METHOD Act_Stop : BOOL
VAR_INPUT
END_VAR
Act_Stop:=stop:=TRUE;
END_METHOD

(*
触发缩回动作，成功触发返回TRUE，触发失败返回FALSE
*)
METHOD Act_Write : BOOL
VAR_INPUT
END_VAR
IF writeStep<10 AND NOT readAndWriteLock THEN
	writeStep:=10;
	readAndWriteLock:=TRUE;
END_IF
END_METHOD

(*
触发缩回动作，成功触发返回TRUE，触发失败返回FALSE
*)
METHOD Act_Write_1 : BOOL
VAR_INPUT
END_VAR
IF writeStep<10 AND readAndWriteLock THEN
	writeStep:=10;
	readAndWriteLock:=TRUE;
END_IF
END_METHOD

ACTION Close_ACT:
//分子泵--close 触发
IF close AND NOT closeCondition THEN
	note_open:=FALSE;
	note_close:=TRUE;
	NoteHMI.showFlag:=TRUE;
	NoteHMI.showText:='';
	NoteHMI.showText:=CONCAT(NoteHMI.showText,nameTXT);
	NoteHMI.showText:=CONCAT(NoteHMI.showText,' Close Condition Not Satisfied!');
	operatorLog.append(CONCAT(nameTXT,' Close Not Done '));
END_IF
IF close AND enable AND closeCondition AND closeStep<20 THEN// AND NOT busy
	note_open:=FALSE;
	note_close:=FALSE;
	busy:=TRUE;
	writeStep:=0;
	writeMaxStep:=0;
	closebusy:=TRUE;
	openbusy:=FALSE;
	open:=FALSE;
	// searial_send(0)**************************************
	opendone:=FALSE;
	closedone:=FALSE;
	openStep:=0;
	closeStep:=10;
	readAndWriteLock:=TRUE;
	PLC_SourceRF.WriteStop();
	operatorLog.append(CONCAT(nameTXT,' Close Done '));
	//errorStep:=0;
END_IF
close:=FALSE;

CASE closeStep OF
0:
	//ready
	
10:
	IF readStep<10 AND writeStep<10 AND writeMaxStep<10 THEN
		closeErrorDelayTon(IN:=FALSE);
		closeDoneDelayTon(IN:=FALSE);
		closeRelay:=TRUE;
		PLC_SourceRF.WriteStop();
		openRelay:=FALSE;
		closeStep:=15;
		t2(IN:=FALSE);
	END_IF
15:
	t2(IN:=TRUE,PT:=T#0.2S);
	IF t2.Q THEN
		t2(IN:=FALSE);
		readAndWriteLock:=FALSE;
		PLC_SourceRF.WriteStop();
		closeStep:=20;
		busy:=FALSE;
	END_IF
20:// DCC与ACC一样，只不过ACC在Open逻辑；DCC 在Close逻辑里；  DCC=forwardpower<setpoint
	closeErrorDelayTon(IN:=(NOT (forwardpower=0 AND reflectedpower=0 AND rematime=0)),PT:=errorDelayTime);
	IF closeErrorDelayTon.Q THEN
		//done:=FALSE;
		opendone:=FALSE;
		closedone:=FALSE;
		errorStep:=2;
		closeStep:=40;
		RETURN;
	END_IF
	IF enablecloseAprSw THEN
		closeDoneDelayTon(IN:=(forwardpower=0 AND reflectedpower=0 AND rematime=0),PT:=doneDelayTimeShortcloseract);
	END_IF
	IF closeDoneDelayTon.Q THEN
		closeErrorDelayTon(IN:=FALSE);
		closeDoneDelayTon(IN:=FALSE);
		closeStep:=30;
	END_IF
30:
	busy:=FALSE;
	closebusy:=FALSE;
	openbusy:=FALSE;
	//done:=TRUE;
	opendone:=FALSE;
	closedone:=TRUE;
	errorStep:=0;
	closeStep:=0;
	readAndWriteLock:=FALSE;
	t2(IN:=FALSE);
40:
	busy:=FALSE;
	closebusy:=FALSE;
	openbusy:=FALSE;
	closeStep:=0;
	readAndWriteLock:=FALSE;
	t2(IN:=FALSE);
END_CASE
END_ACTION

ACTION Error_ACT:
CASE errorStep OF
	0:
		error:=FALSE;
		errID:=0;
		errTXT:='';
 (*
	1:
		error:=TRUE;
		errID:=errorID+errorStep;
		errTXT:=CONCAT(STR1:=nameTXT,STR2:=' Extend Error!');
		errWTXT:=WCONCAT(STR1:=TO_WSTRING(nameTXT),STR2:=" 伸出(打开)错误");
	2:
		error:=TRUE;
		errID:=errorID+errorStep;
		errTXT:=CONCAT(STR1:=nameTXT,STR2:=' Retract Error!');
		errWTXT:=WCONCAT(STR1:=TO_WSTRING(nameTXT),STR2:=" 缩回(关闭)错误");
		*)
	1..6:
		error:=TRUE;
		errID:=getErrID(errorStep);
		errTXT:=getErrTXT(errorStep);
		errWTXT:=getErrWTXT(errorStep);
END_CASE
END_ACTION

METHOD Get_Done_Close : BOOL
VAR_INPUT
END_VAR
Get_Done_Close:=closedone;
END_METHOD

METHOD Get_Done_Open : BOOL
VAR_INPUT
END_VAR
Get_Done_Open:=opendone;
END_METHOD

METHOD getErrID : UDINT
VAR_INPUT
	errID					:UDINT;//取值范围1~2
END_VAR
VAR
	nErrID					:UDINT;
END_VAR
nErrID:=errorID+errID;

getErrID:=nErrID;
END_METHOD

METHOD getErrTXT : STRING(255)
VAR_INPUT
	errID					:UDINT;//取值范围1~2
END_VAR
VAR
	sErrTXT					:STRING(255);
END_VAR

CASE errID OF
	1:
		sErrTXT:=CONCAT(STR1:=nameTXT,STR2:=' Open(TimeOut) Error!');
	2:
		sErrTXT:=CONCAT(STR1:=nameTXT,STR2:=' Close Error!');
	3:
		sErrTXT:=CONCAT(STR1:=nameTXT,STR2:=' NormalRun Error!');
	4:
		sErrTXT:=CONCAT(STR1:=nameTXT,STR2:=' CheckCondition Error!');
	5:
		sErrTXT:=CONCAT(STR1:=nameTXT,STR2:=' ParSet Fault!');
	6:
		sErrTXT:=CONCAT(STR1:=nameTXT,STR2:=' Communication Error!');
ELSE
	sErrTXT:=CONCAT(STR1:=nameTXT,STR2:='');
END_CASE
getErrTXT:=sErrTXT;
END_METHOD

METHOD getErrWTXT : WSTRING(255)
VAR_INPUT
	errID					:UDINT;//取值范围1~16
END_VAR
VAR
	sErrTXT					:WSTRING(255);
END_VAR

CASE errID OF
	1:
		sErrTXT:=WCONCAT(STR1:=TO_WSTRING(nameTXT),STR2:=" RF启动错误");
	2:
		sErrTXT:=WCONCAT(STR1:=TO_WSTRING(nameTXT),STR2:=" RF停止错误");
	3:
		sErrTXT:=WCONCAT(STR1:=TO_WSTRING(nameTXT),STR2:=" RF正常运行出现异常情况");
	4:
		sErrTXT:=WCONCAT(STR1:=TO_WSTRING(nameTXT),STR2:=" 检测到条件异常，关机处理");
	5:
		sErrTXT:=WCONCAT(STR1:=TO_WSTRING(nameTXT),STR2:=" 参数设置有误");
	6:
		sErrTXT:=WCONCAT(STR1:=TO_WSTRING(nameTXT),STR2:=" 通讯异常");
		
ELSE
	sErrTXT:=WCONCAT(STR1:=TO_WSTRING(nameTXT),STR2:="");
END_CASE
getErrWTXT:=sErrTXT;
END_METHOD

ACTION Init_ACT:
done:=(opendone OR closedone);
powerTon(IN:=mainPower,PT:=T#10S);
IF AlmAprSw AND powerTon.Q THEN
	errorStep:=5;
END_IF
IF readerror OR NOT readCondition AND firstPowerTON.Q THEN
	errorStep:=6;
END_IF
error:=error OR serialError OR NOT mainPower OR AlmAprSw;
InitHMI_ACT();
manualCtrl_ACT();
IF (error OR AlmAprSw OR ErrorAprSw OR NOT openCondition) AND openRelay THEN
	stop:=TRUE;
	busy:=FALSE;
	openRelay:=FALSE;
END_IF

noteTON_P(IN:=note_open,PT:=T#0.1S);
noteRTrig_P(CLK:=noteTON_P.Q);
IF noteRTrig_P.Q THEN
//	gLog_Note.append_EX(noteWTXT_Open);
END_IF
noteTON_N(IN:=note_close,PT:=T#0.1S);
noteRTrig_N(CLK:=noteTON_N.Q);
IF noteRTrig_N.Q THEN
//	gLog_Note.append_EX(noteWTXT_close);
END_IF
END_ACTION

ACTION InitHMI_ACT:
HMIItf.AlmAprSw:=AlmAprSw;
HMIItf.ErrorAprSw:=ErrorAprSw;

HMIItf.temperature:=temperature;
HMIItf.current:=current;
HMIItf.vol:=vol;

HMIItf.enableOpen:=enableOpenAprSw;
HMIItf.enableClose:=enableCloseAprSw;
HMIItf.HMIEnable:=hmiEN;
HMIItf.enable:=enable;
HMIItf.done:=done;
HMIItf.busy:=busy;
HMIItf.error:=error;
HMIItf.errID:=UDINT_TO_DINT(errID);
HMIItf.errTXT:=errTXT;
HMIItf.openRelay:=openRelay;
HMIItf.resetRelay:=resetRelay;

HMIItf.power:=power;
HMIItf.nameTXT:=nameTXT;

HMIItf.runTime:=runTime;
HMIItf.opencondition:=openCondition;
HMIItf.closecondition:=closeCondition;
END_ACTION

ACTION ManualCtrl_ACT:
//HMI手动控制
//IF ctrlMode=eManualCtrMode THEN
IF hmiEN THEN
	extendTrigRAlc(CLK:=HMIItf.extendAndretract);
	IF extendTrigRAlc.Q THEN// AND NOT busy
		IF openRelay THEN// 如果启动继电器或全速，则认为已经已启动完毕
			close:=TRUE;
		END_IF
		IF NOT openRelay THEN
			open:=TRUE;
		END_IF
	END_IF
	openendTrigR1_Aiko(CLK:=HMIItf.bopen);
	IF openendTrigR1_Aiko.Q AND NOT busy AND NOT openRelay THEN
		open:=TRUE;
		close:=FALSE;
	END_IF
	IF openendTrigR1_Aiko.Q AND busy AND openRelay THEN
		close:=TRUE;
		open:=FALSE;
	END_IF
	
	singleControltempR(CLK:=HMIItf.singleControltemp);
	openendTrigR1(CLK:=HMIItf.open);
	IF openendTrigR1.Q OR (singleControltempR.Q AND NOT openRelay ) THEN// AND NOT busy
		WarmHMI.showText:='';
		WarmHMI.showFlag:=TRUE;
		WarmHMI.showText:=CONCAT(WarmHMI.showText,'Are you sure you want to Open the ');
		WarmHMI.showText:=CONCAT(WarmHMI.showText,nameTXT);
		WarmHMI.showText:=CONCAT(WarmHMI.showText,' ?');
	END_IF
	IF WarmHMI.bOK AND NOT WarmHMI.showFlag AND FIND(WarmHMI.showText,nameTXT)>0 AND FIND(WarmHMI.showText,'Open')>0 THEN
		open:=TRUE;
		operatorLog.append(CONCAT(CONCAT(nameTXT,' Open:'),UDINT_TO_STRING(setpower)));
		operatorLog.append(CONCAT(CONCAT(nameTXT,' Open:'),UDINT_TO_STRING(settime)));
		WarmHMI.bOK:=FALSE;
		WarmHMI.showText:='';
	END_IF
	IF WarmHMI.bNO AND NOT WarmHMI.showFlag AND FIND(WarmHMI.showText,nameTXT)>0 AND FIND(WarmHMI.showText,'Open')>0 THEN
		WarmHMI.bNO:=FALSE;
		WarmHMI.showText:='';
	END_IF
	
	closeractTrigR1(CLK:=HMIItf.close);
	IF closeractTrigR1.Q OR (singleControltempR.Q AND openRelay) THEN// AND NOT busy
		WarmHMI.showText:='';
		WarmHMI.showFlag:=TRUE;
		WarmHMI.showText:=CONCAT(WarmHMI.showText,'Are you sure you want to Close the ');
		WarmHMI.showText:=CONCAT(WarmHMI.showText,nameTXT);
		WarmHMI.showText:=CONCAT(WarmHMI.showText,' ?');
	END_IF
	IF WarmHMI.bOK AND NOT WarmHMI.showFlag AND FIND(WarmHMI.showText,nameTXT)>0 AND FIND(WarmHMI.showText,'Close')>0 THEN
		close:=TRUE;
		operatorLog.append(CONCAT(nameTXT,' Close'));
		WarmHMI.bOK:=FALSE;
		WarmHMI.showText:='';
	END_IF
	IF WarmHMI.bNO AND NOT WarmHMI.showFlag AND FIND(WarmHMI.showText,nameTXT)>0 AND FIND(WarmHMI.showText,'Close')>0 THEN
		WarmHMI.bNO:=FALSE;
		WarmHMI.showText:='';
	END_IF
	
	resetTrigR1(CLK:=HMIItf.reset);
	IF resetTrigR1.Q THEN// AND NOT busy
		reset:=TRUE;
	END_IF
	
	stopTrigR1(CLK:=HMIItf.stop);
	IF stopTrigR1.Q THEN// AND NOT busy
		stop:=TRUE;
	END_IF
	
	powerTrigR1(CLK:=HMIItf.power);
	IF powerTrigR1.Q THEN// AND NOT busy
		IF power THEN
			power:=FALSE;
		ELSE
			power:=TRUE;
		END_IF
	END_IF
	
END_IF
END_ACTION

ACTION Open_ACT:
//分子泵伸出--open 触发
IF open AND NOT openCondition THEN
	note_open:=TRUE;
	note_close:=FALSE;
	NoteHMI.showFlag:=TRUE;
	NoteHMI.showText:='';
	NoteHMI.showText:=CONCAT(NoteHMI.showText,nameTXT);
	NoteHMI.showText:=CONCAT(NoteHMI.showText,' Open Condition Not Satisfied!');
	operatorLog.append(CONCAT(nameTXT,' Open Not Done '));
END_IF
IF open AND enable AND openCondition AND NOT AlmAprSw AND NOT ErrorAprSw AND NOT openbusy AND mainPower AND NOT resetRelay THEN// AND NOT busy
	note_open:=FALSE;
	note_close:=FALSE;
	busy:=TRUE;
	closebusy:=FALSE;
	openbusy:=TRUE;
	close:=FALSE;
	open:=FALSE;
	done:=FALSE;
	opendone:=FALSE;
	closedone:=FALSE;
	openStep:=10;
	writeStep:=0;
	writeMaxStep:=0;
	readAndWriteLock:=TRUE;
	// searial_send(setPoint)**************************************
	closeStep:=0;
	operatorLog.append(CONCAT(nameTXT,' Open Done '));
END_IF
open:=FALSE;
runTimeClearR(CLK:=HMIItf.runTimeClear);
runTON(IN:=NOT error AND openRelay AND NOT runTON.Q, PT:=T#60S);// 1小时计数一次,启动，无报错，且全速
IF runTON.Q AND runTime<999999999999999 AND NOT runTimeClearR.Q THEN
	runTime:=runTime+1;
END_IF
IF runTimeClearR.Q THEN
	runTime:=0;
END_IF
//IF NOT openRelay AND NOT AccAprSw AND NOT DccAprSw AND NOT NormalAprSw THEN// 计数清零
//	runTime:=0;
//END_IF

CASE openStep OF
0:
	//ready
	runTON(IN:=FALSE);
	openErrorDelayTon(IN:=FALSE);
	openErrorDelayTon(IN:=FALSE);
	openDoneDelayTon(IN:=FALSE);
	t1(IN:=FALSE);
	rematime:=0;
10:
	IF setpower<1 OR (NOT co_control AND settime<1) THEN 
		open:=FALSE;
		close:=FALSE;
		openbusy:=FALSE;
		closebusy:=FALSE;
		errorStep:=5;
		openStep:=60;
	ELSE
		t1(IN:=readStep<10 AND writeStep<10 AND writeMaxStep<10,PT:=T#0.5S);
		IF t1.Q THEN
			openErrorDelayTon(IN:=FALSE);
			openDoneDelayTon(IN:=FALSE);
			openStep:=15;
			openRelay:=TRUE;
			setpointdone:=FALSE;
			Act_Write_1();
			openbusy:=TRUE;
			closebusy:=FALSE;
			closeRelay:=FALSE;
			t1(IN:=FALSE);
		END_IF
	END_IF
15:
	t1(IN:=setpointdone,PT:=T#0.1S);
	IF t1.Q THEN
		setpointdone:=FALSE;
		t1(IN:=FALSE);
		PLC_SourceRF.receiveFlag:=FALSE;
		PLC_SourceRF.WriteStart();
		openStep:=17;
	END_IF
17:
	t1(IN:=PLC_SourceRF.receiveFlag,PT:=T#0.05S);
	IF t1.Q THEN
		t1(IN:=FALSE);
		PLC_SourceRF.receiveFlag:=FALSE;
		readAndWriteLock:=FALSE;
		busy:=false;
		openStep:=20;
	END_IF
20:
	// AccAprSw可以看成是forward Power > 5 ,< set point - 5// 或者反射功率>0
	openErrorDelayTon(IN:=(NOT (ABS(forwardpower)>=0 AND reflectedpower<10 AND ABS(setpower-forwardpower)<2)),PT:=errorDelayTime);
	IF openErrorDelayTon.Q THEN
		//done:=FALSE;
		open:=FALSE;
		close:=FALSE;
		openbusy:=FALSE;
		closebusy:=FALSE;
		errorStep:=1;
		openStep:=60;
		RETURN;
	END_IF
	IF enableopenAprSw THEN
		openDoneDelayTon(IN:=ABS(forwardpower)>=0 AND reflectedpower<10 AND ABS(setpower-forwardpower)<2,PT:=doneDelayTimeShortopenend);
	END_IF
	IF openDoneDelayTon.Q THEN
		openErrorDelayTon(IN:=FALSE);
		openDoneDelayTon(IN:=FALSE);
		openStep:=30;
	END_IF
	
	//状态实时检测
	IF NOT openCondition AND (NOT closedone OR openRelay) THEN// 检测到开条件消失，强制关闭
		openRelay:=FALSE;
		errorStep:=4;
		openbusy:=FALSE;
		closebusy:=FALSE;
		openStep:=60;
	END_IF
	IF (ErrorAprSw OR AlmAprSw) AND openRelay THEN//只要报错；启动线圈启动，强锁启动信号
		openRelay:=FALSE;
		openStep:=60;/////
		errorStep:=3;
		openbusy:=FALSE;
		closebusy:=FALSE;
	END_IF
30:
	openErrorDelayTon(IN:=NOT co_control,PT:=UDINT_TO_TIME(settime*1000));// 反射调整超时时间
	rematime:=TIME_TO_UDINT(openErrorDelayTon.ET/1000);
	rematime:=settime-rematime;
	IF openErrorDelayTon.Q OR co_control THEN
		openStep:=40;
		rematime:=0;
		openErrorDelayTon(IN:=FALSE);
	END_IF
	// 状态实时检测
	IF NOT openCondition AND (NOT closedone OR openRelay) THEN//蝶阀单控，检测到开条件消失，强制关闭
		openRelay:=FALSE;
		errorStep:=4;
		openStep:=60;
		closebusy:=FALSE;
		openbusy:=FALSE;
	END_IF
	IF (ErrorAprSw OR AlmAprSw) AND openRelay THEN//只要报错；启动线圈启动，强锁启动信号
		openRelay:=FALSE;
		stop:=TRUE;
		openStep:=60;/////
		errorStep:=3;
		closebusy:=FALSE;
		openbusy:=FALSE;
	END_IF
40:
	busy:=FALSE;
	IF NOT co_control THEN
		openRelay:=FALSE;
		close:=TRUE;
	END_IF
	openStep:=50;
	openbusy:=FALSE;
	readAndWriteLock:=FALSE;
	opendone:=TRUE;
50:
	rematime:=0;
60:
	openRelay:=FALSE;
	openStep:=70;
	busy:=FALSE;
	readAndWriteLock:=FALSE;
	;//报错
	co_control:=FALSE;
	opendone:=FALSE;
END_CASE
END_ACTION

ACTION Read_ACT:
//气缸收回--read 触发
firstPowerTON(IN:=firstPower,PT:=T#10S);
readTON(IN:=NOT readAndWriteLock AND NOT busy AND NOT readbusy AND readStep=0 AND readCondition,PT:=T#0.05S);
IF readTON.Q THEN// AND NOT busy
	readdone:=FALSE;
	readStep:=10;
	readbusy:=TRUE;
	readerror:=FALSE;
END_IF
CASE readStep OF
0:
	//ready
	readTon1(IN:=FALSE);
	readTon2(IN:=FALSE);
	readTon3(IN:=FALSE);
10:// State
	IF gICP.SourceRF.controlMode=2 THEN
		PLC_SourceRF.readStateFlag:=FALSE;
		PLC_SourceRF.ReadState();
		readStep:=readStep+10;
	ELSE
		PLC_SourceRF.readStateFlag:=FALSE;
		PLC_SourceRF.WriteRS232Mode();
		readStep:=readStep+15;
		PLC_SourceRF.receiveFlag:=FALSE;
	END_IF
20:
	IF PLC_SourceRF.readStateFlag THEN
		PLC_SourceRF.readStateFlag:=FALSE;
		// 数据处理
		readTon1(IN:=FALSE);
		readStep:=readStep+10;
		RETURN;
	END_IF
	readTon1(IN:=TRUE,PT:=T#500MS);// 超时
	IF readTon1.Q THEN
		readStep:=6000;
		readTon1(IN:=FALSE);
		readTon2(IN:=FALSE);
		RETURN;
	END_IF
25:
	IF PLC_SourceRF.receiveFlag THEN
		PLC_SourceRF.receiveFlag:=FALSE;
		// 数据处理
		readTon1(IN:=FALSE);
		readStep:=readStep+5;
		RETURN;
	END_IF
	readTon1(IN:=TRUE,PT:=T#500MS);// 超时
	IF readTon1.Q THEN
		readStep:=6000;
		readTon1(IN:=FALSE);
		readTon2(IN:=FALSE);
		RETURN;
	END_IF
30:
	readTon3(IN:=TRUE,PT:=T#0.1S);
	IF readTon3.Q THEN
		readStep:=readStep+10;
		readTon3(IN:=FALSE);
	END_IF
40:// State
	PLC_SourceRF.readStateFlag:=FALSE;
	PLC_SourceRF.ReadState();
	readStep:=readStep+10;
50:
	IF PLC_SourceRF.readStateFlag THEN
		PLC_SourceRF.readStateFlag:=FALSE;
		// 数据处理
		readTon1(IN:=FALSE);
		readStep:=readStep+10;
		RETURN;
	END_IF
	readTon1(IN:=TRUE,PT:=T#500MS);// 超时
	IF readTon1.Q THEN
		readStep:=6000;
		readTon1(IN:=FALSE);
		readTon2(IN:=FALSE);
		RETURN;
	END_IF
60:
	readStep:=90;
90:
	readTon3(IN:=TRUE,PT:=T#0.1S);
	IF readTon3.Q THEN
		readStep:=5000;
		readTon3(IN:=FALSE);
	END_IF
5000:
	readbusy:=FALSE;
	readdone:=TRUE;
	readStep:=0;
	readerror:=FALSE;
	PLC_SourceRF.ClearCom:=TRUE;
6000:
	readbusy:=FALSE;
	readdone:=TRUE;
	readStep:=0;
	readErrorTimes:=readErrorTimes+1;
	IF readErrorTimes>3 THEN
		readErrorTimes:=0;
		readerror:=TRUE;
		gICP.SourceRF.setpowerRead:=0;
		gICP.SourceRF.forwardpower:=0;
		gICP.SourceRF.reflectedpower:=0;
		gICP.SourceRF.maxpower:=0;
	END_IF
	gICP.SourceRF.controlMode:=0;
END_CASE
END_ACTION

ACTION Reset_ACT:
IF reset THEN
	IF NOT power THEN
		openRelay:=FALSE;
		closeRelay:=FALSE;
	END_IF
	note_open:=FALSE;
	note_close:=FALSE;
	IF errorStep<>0 OR  AlmAprSw OR ErrorAprSw THEN
		errorStep:=0;
		busy:=FALSE;
		closebusy:=FALSE;
		openbusy:=FALSE;
		resetRelay:=TRUE;
		readAndWriteLock:=TRUE;
		PLC_SourceRF.WriteReset();
	END_IF
	reset:=FALSE;
	note_open:=FALSE;
	note_close:=FALSE;
END_IF
resetRelayTON(IN:=resetRelay , PT:=resetRelayTONTime);
IF resetRelayTON.Q THEN
	errorStep:=0;
	busy:=FALSE;
	resetRelay:=FALSE;
	readAndWriteLock:=FALSE;
END_IF

IF stop THEN
	note_open:=FALSE;
	note_close:=FALSE;
	stop:=FALSE;
	openRelay:=FALSE;
	closeRelay:=FALSE;
	//无自锁检测说法，直接停
	openStep:=0;
	closeStep:=0;
	writeStep:=0;
	writeMaxStep:=0;
END_IF
END_ACTION

ACTION VersionLog:
(*
版本: V1.0.0.0
说明:
	1. 首个版本
	2. 含普通分子泵\泵组类型的控制
	3. 可配置是否有到位信号, 以及到位稳定时间
(--------------------------------------------------)
新版本: V1.0.1.0
更新时间: 2019/11/20 19:00
更新说明:
	1. 优化编写方式
	2. 修改错误编码起始位，现改为从1开始
(--------------------------------------------------)
新版本: V1.0.1.1
更新时间: 2020/03/23 23:00
更新说明:
	1. 优化报错方式
	2. 增加伸出、缩回、复位和停止触发函数
(--------------------------------------------------)
新版本: V1.0.1.2
更新时间: 2020/04/22 09:50
更新说明:
	1. 增加中文报警输出
(--------------------------------------------------)
新版本: V1.0.1.3
更新时间: 2020/09/16
更新说明:
	1. 开放错误ID、错误文本信息获取接口
(--------------------------------------------------)
新版本: V1.0.1.4
更新时间: 2020/10/06
更新说明:
	1. 移除控制模式变量，增加HMI启用条件
	2. 增加外部获取伸出缩回完成信号接口函数
(--------------------------------------------------)
新版本: V1.0.1.5
更新时间: 2020/10/14
更新说明:
	1. 优化代码
(--------------------------------------------------)
新版本: V2.0.1.0
更新时间: 2023/11/17
更新说明:
	1. 分子泵控制独立
(--------------------------------------------------)


*)
END_ACTION

ACTION WriteMaxPower_ACT:
//分子泵--write 触发

CASE writeMaxStep OF
0:
	//ready
	writeMaxTON(IN:=FALSE);
10:
	readAndWriteLock:=TRUE;
	writeMaxTON(IN:=TRUE,PT:=T#3S);
	IF writeMaxTON.Q THEN
		writeMaxTON(IN:=FALSE);
		writeMaxStep:=writeMaxStep+10;
	END_IF
20:
	IF readStep<10 AND openStep<10 AND closeStep<10 AND writeStep<10 THEN
		PLC_SourceRF.WriteMaxPower(gICP.SourceRF.setpower);
		writeMaxStep:=writeMaxStep+10;
	END_IF
30:
	writeMaxTON(IN:=TRUE,PT:=T#3S);
	IF writeMaxTON.Q THEN
		writeMaxTON(IN:=FALSE);
		writeMaxStep:=writeMaxStep+10;
	END_IF
40:
	writeMaxStep:=100;
100:
	writeMaxStep:=0;	
	readAndWriteLock:=FALSE;
END_CASE
END_ACTION

ACTION WritePower_ACT:
//分子泵--write 触发

CASE writeStep OF
0:
	//ready
	writeTON(IN:=FALSE);
10:
	writeTON(IN:=readStep<10,PT:=T#0.1S);
	setpointdone:=FALSE;
	IF writeTON.Q THEN
		PLC_SourceRF.ClearCom:=TRUE;
		writeTON(IN:=FALSE);
		writeStep:=writeStep+10;
	END_IF
20:
	IF readStep<10  AND writeMaxStep<10 THEN
		PLC_SourceRF.WritePower(gICP.SourceRF.setpower);
		PLC_SourceRF.receiveFlag:=FALSE;
		writeStep:=writeStep+10;
	END_IF
30:
	writeTON(IN:=NOT PLC_SourceRF.receiveFlag ,PT:=T#0.5S);
	IF writeTON.Q THEN
		PLC_SourceRF.receiveFlag:=FALSE;
		writeTON(IN:=FALSE);
		writeStep:=writeStep+10;
		setpointdone:=FALSE;
		RETURN;
	END_IF
	IF PLC_SourceRF.receiveFlag THEN
		PLC_SourceRF.receiveFlag:=FALSE;
		writeTON(IN:=FALSE);
		writeStep:=writeStep+10;
		setpointdone:=TRUE;
		RETURN;
	END_IF
40:
	writeStep:=100;
100:
	writeStep:=0;	
	readAndWriteLock:=FALSE;
END_CASE
END_ACTION

END_FUNCTION_BLOCK

// ---- POUs/Communication/PLC_SourceRF.TcPOU
PROGRAM PLC_SourceRF
PROGRAM PLC_SourceRF
VAR_INPUT
	nSocketType:UINT:=0;// socket 类型; 0 表示 server; 1 表示 client;
	sTerminalName:STRING;// 通讯对方名称 自定义
	sHost:STRING(20):='127.0.0.1';// 通讯IP地址; server时表示本地host; client时表示远程host
	nPort:UDINT:=8900;// 通讯端口号;
	bEnable:BOOL:=TRUE;// 通讯启用\禁用连接
	sSendSuffix:STRING:='';//此处可统一添加发送后缀字符 $R$N
	nQueueInterval:UDINT:=50;// 发送队列时间间隔 单位ms
	logHandleArray:ARRAY [1..5] OF POINTER TO printLogModule_EX;// log 操作 handle 数组
	logHandleArrayLength:UINT:=0;// log 操作 handle 数组长度, 不超过5
	readStateFlag:BOOL;
	ClearCom:BOOL;
	receiveFlag:BOOL;
END_VAR
VAR_OUTPUT
	bSendCondition	:BOOL;//可发送条件
	bSocketConnected:BOOL;//连接状态
END_VAR
VAR CONSTANT
	cNumBegin		:DINT:=1;
	cNumEnd			:DINT:=100;
END_VAR
VAR
	sendDataArray	:ARRAY [cNumBegin..cNumEnd] OF STRING(255);
	length			:DINT:=0;
	endPoint		:DINT:=cNumBegin;
	popupSendData	:STRING(255);
	//popup
	popupStep		:UINT:=0;
	popupTON1		:TON;
	popupTON2		:TON;
	iPopup			:DINT:=0;
	_PopupLength	:DINT:=0;
END_VAR
VAR
	tcpipClient					:tcpipClientModule_EX;
	tcpipServer					:tcpipServerModule_EX;////定义服务器对象
	
	tcpipSendDataBuff_Server	:STRING(255);//发送数据 Buff server
	tcpipSendDataBuff_Client	:STRING(255);//发送数据 Buff client
	
	tcpipSendDataClear			:STRING(255);//发送数据 清空
	tcpipSendData				:STRING(255);//发送数据
	
	tcpipRecDataBuff_Server		:STRING(255);//已接收数据 Buff server
	tcpipRecDataBuff_Client		:STRING(255);//已接收数据 Buff client
	
	tcpipRecDataClear			:STRING(255);//已接收数据 清空
	tcpipRecData				:STRING(255);//已接收数据
	
	tcpConnectR_Trig			:R_Trig;//初始连接上升沿
	tcpConnectF_Trig			:F_Trig;//初始连接下降沿
	registerStep				:UDINT;//ALC注册控制步
	registerTON					:TON;//ALC注册延时
	
	logHandleArray_index		:UINT:=1;
END_VAR
VAR
	bTrig_Start:BOOL;
	rTrig_Start:R_TRIG;
	tTrig_Start:TON;
	
	bTrig_Stop:BOOL;
	rTrig_Stop:R_TRIG;
	tTrig_Stop:TON;
	
	bTrig_Reset:BOOL;
	rTrig_Reset:R_TRIG;
	tTrig_Reset:TON;
	
	
	bTrig_Init:BOOL;
	rTrig_Init:R_TRIG;
	
	bTrig_All_Home:BOOL;
	rTrig_All_Home:R_TRIG;
	
	bTrig_Z_Safe:BOOL;
	rTrig_Z_Safe:R_TRIG;
	
	bTrig_P_Pos_:BOOL;
	rTrig_P_Pos_:R_TRIG;
	nTrig_P_Pos_TrayNum:UINT:=1;
	nTrig_P_Pos_RowNum:UINT:=1;
	
	bTrig_Move_P_:BOOL;
	rTrig_Move_P_:R_TRIG;
	nTrig_Move_P_TrayNum:UINT:=1;
	nTrig_Move_P_RowNum:UINT:=1;
	nTrig_Move_P_PosNum:UINT:=1;
	findposstart	:INT;
	findposend		:INT;
	find_pos		:INT;
	recStrTemp		:STRING(255);
END_VAR


CASE nSocketType OF
0://TCPIP server
	tcpipServer(
		sSrvNetId:= , 
		sLocalHost:=sHost , 
		nLocalPort:=nPort , 
		bStartConnect:=bEnable , 
		tcpipSDataLen:=TO_UDINT(LEN(tcpipSendDataBuff_Server)) , 
		tcpipSData:=ADR(tcpipSendDataBuff_Server) , 
		bSend:= , 
		tcpipRecDataLen:=SIZEOF(tcpipRecDataBuff_Server) , 
		tcpipRecData:=ADR(tcpipRecDataBuff_Server) , 
		bAccepted=> , 
		bSendBusy=> , 
		bRecData=> );
	bSendCondition:=tcpipServer.bAccepted AND NOT tcpipServer.bSendBusy;
	//TCPIP连接
	bSocketConnected:=tcpipServer.bAccepted;
	IF NOT tcpipServer.bAccepted THEN
		length:=0;
		endPoint:=cNumBegin;
	END_IF
	tcpConnectR_Trig(CLK:=tcpipServer.bAccepted);
	tcpConnectF_Trig(CLK:=tcpipServer.bAccepted);

1://TCPIP client
	tcpipClient(
		sSrvNetId:= , 
		sRemoteHost:=sHost , 
		nRemotePort:=nPort , 
		bStartConnect:=bEnable , 
		tcpipSDataLen:=TO_UDINT(LEN(tcpipSendDataBuff_Client)) , 
		tcpipSData:=ADR(tcpipSendDataBuff_Client) , 
		bSend:= , 
		tcpipRecDataLen:=SIZEOF(tcpipRecDataBuff_Client) , 
		tcpipRecData:=ADR(tcpipRecDataBuff_Client) , 
		bConnected=> , 
		bSendBusy=> , 
		bRecData=> );
	bSendCondition:=tcpipClient.bConnected AND NOT tcpipClient.bSendBusy;
	//TCPIP连接
	bSocketConnected:=tcpipClient.bConnected;
	IF NOT tcpipClient.bConnected THEN
		length:=0;
		endPoint:=cNumBegin;
	END_IF
	tcpConnectR_Trig(CLK:=tcpipClient.bConnected);
	tcpConnectF_Trig(CLK:=tcpipClient.bConnected);
END_CASE
IF ClearCom THEN
	length:=0;
	endPoint:=cNumBegin;
	ClearCom:=FALSE;
END_IF
IF tcpConnectR_Trig.Q THEN
	FOR logHandleArray_index:=1 TO logHandleArrayLength DO
		logHandleArray[logHandleArray_index]^.append(CONCAT(sTerminalName, ' has been connected'));
	END_FOR
	registerStep:=10;
END_IF
IF tcpConnectF_Trig.Q THEN
	FOR logHandleArray_index:=1 TO logHandleArrayLength DO
		logHandleArray[logHandleArray_index]^.append(CONCAT(sTerminalName, ' has been disconnected'));
	END_FOR
	registerStep:=0;
END_IF
//数据接收处理
CASE nSocketType OF
0://TCPIP server
	IF tcpipServer.bRecData THEN
		tcpipRecData:=tcpipRecDataBuff_Server;//buff转存
		tcpipRecDataBuff_Server:=tcpipRecDataClear;//转存之后清空buff
		dataProcessing();
	END_IF
1://TCPIP client
	IF tcpipClient.bRecData THEN
		tcpipRecData:=tcpipRecDataBuff_Client;//buff转存
		tcpipRecDataBuff_Client:=tcpipRecDataClear;//转存之后清空buff
		dataProcessing();
	END_IF
END_CASE


popup();

CASE registerStep OF
0:
	//Ready
END_CASE

METHOD appendSend : BOOL
VAR_INPUT
	str			:STRING(255);
END_VAR
VAR
	suffix					:STRING;
	strTemp_appendSend		:STRING(255);
END_VAR

IF endPoint>(cNumEnd-1) THEN
	RETURN;
END_IF
suffix:=sSendSuffix;//此处可统一添加发送后缀字符 $R$N

strTemp_appendSend:=CONCAT(str,suffix);
sendDataArray[endPoint]:=strTemp_appendSend;

endPoint:=endPoint+1;
length:=endPoint-cNumBegin;
END_METHOD

METHOD dataProcessing : BOOL
VAR_INPUT
END_VAR
VAR
	strTemp:STRING;
END_VAR
FOR logHandleArray_index:=1 TO logHandleArrayLength DO
	CASE nSocketType OF
	0://TCPIP server
//		logHandleArray[logHandleArray_index]^.append(CONCAT(CONCAT(CONCAT('Recevie From ', sTerminalName), ' -- '),tcpipRecData));
	1://TCPIP client
//		logHandleArray[logHandleArray_index]^.append(CONCAT(CONCAT(CONCAT('Recevie From ', sTerminalName), ' -- '),tcpipRecData));
	END_CASE
END_FOR
receiveFlag:=TRUE;
findposend:=0;
find_pos:=0;
IF MID(tcpipRecData,1,32)='$R' AND MID(tcpipRecData,1,33)='$R'  THEN
	gICP.SourceRF.controlMode:=STRING_TO_INT(MID(tcpipRecData,1,1));
	gICP.SourceRF.outputMode:=STRING_TO_INT(MID(tcpipRecData,1,2));
	gICP.SourceRF.outputState:=STRING_TO_INT(MID(tcpipRecData,1,3));
	strTemp:='';
	strTemp:=CONCAT(strTemp,(MID(tcpipRecData,2,6)));
	gICP.SourceRF.alarmState:=STRING_TO_INT(strTemp);
	strTemp:='';
	strTemp:=CONCAT(strTemp,(MID(tcpipRecData,5,9)));
	gICP.SourceRF.setpowerRead:=STRING_TO_UDINT(strTemp);
	strTemp:='';
	strTemp:=CONCAT(strTemp,(MID(tcpipRecData,5,15)));
	gICP.SourceRF.forwardpower:=STRING_TO_UDINT(strTemp);
	strTemp:='';
	strTemp:=CONCAT(strTemp,(MID(tcpipRecData,5,21)));
	gICP.SourceRF.reflectedpower:=STRING_TO_UDINT(strTemp);
	strTemp:='';
	strTemp:=CONCAT(strTemp,(MID(tcpipRecData,5,27)));
	gICP.SourceRF.maxpower:=STRING_TO_UDINT(strTemp);
	readStateFlag:=TRUE;
END_IF
END_METHOD

METHOD PRIVATE popup : BOOL
VAR_INPUT
END_VAR
CASE popupStep OF
0:
	IF length>0 AND bSendCondition THEN
		_PopupLength:=length;
		popupSendData:=sendDataArray[cNumBegin];
		FOR iPopup:=cNumBegin TO (_PopupLength-1) DO
			sendDataArray[iPopup]:=sendDataArray[iPopup+1];
		END_FOR
		endPoint:=endPoint-1;
		length:=endPoint-cNumBegin;
		sendData(popupSendData);//此处是调用信息发送
		popupStep:=10;
	END_IF
10:
	popupTON2(IN:=NOT popupTON2.Q, PT:=T#2S);
	IF NOT bSendCondition OR popupTON2.Q THEN
		popupTON2(IN:=FALSE);
		popupStep:=11;
	END_IF
11:
	IF bSendCondition THEN
		popupStep:=12;
	END_IF
	popupTON1(IN:=FALSE);
12:
	//popupTON1(IN:=NOT popupTON1.Q,PT:=T#10MS);
	popupTON1(IN:=NOT popupTON1.Q,PT:=TO_TIME(nQueueInterval));
	IF popupTON1.Q THEN
		popupStep:=0;
	END_IF
END_CASE
END_METHOD

METHOD ReadState : BOOL
VAR_INPUT
END_VAR
VAR
END_VAR
appendSend('Q$R');
END_METHOD

METHOD PRIVATE sendData : BOOL
VAR_INPUT
	dataStruct	:STRING(255);
END_VAR
IF bSendCondition AND bEnable THEN
	tcpipSendData:=dataStruct;
	
	CASE nSocketType OF
	0://TCPIP server
		tcpipSendDataBuff_Server:=tcpipSendData;
		tcpipSendData:=tcpipSendDataClear;	
		tcpipServer.bSend:=TRUE;
	1://TCPIP client
		tcpipSendDataBuff_Client:=tcpipSendData;
		tcpipSendData:=tcpipSendDataClear;	
		tcpipClient.bSend:=TRUE;
	END_CASE
	
	FOR logHandleArray_index:=1 TO logHandleArrayLength DO
		CASE nSocketType OF
		0://TCPIP server
//			logHandleArray[logHandleArray_index]^.append(CONCAT(CONCAT(CONCAT('Send To ', sTerminalName), ' -- '),tcpipSendDataBuff_Server));
		1://TCPIP client
//			logHandleArray[logHandleArray_index]^.append(CONCAT(CONCAT(CONCAT('Send To ', sTerminalName), ' -- '),tcpipSendDataBuff_Client));
		END_CASE
	END_FOR
END_IF
END_METHOD

METHOD WriteMaxPower : BOOL
VAR_INPUT
	maxpowerpoint:UDINT;
END_VAR
VAR
	str:STRING;
	_bit:UDINT;
	_ten:UDINT;
	_hundred:UDINT;
	_thousand:UDINT;
END_VAR
str:='';
_thousand:=maxpowerpoint/1000;
str:=CONCAT(str,UDINT_TO_STRING(maxpowerpoint));
//_hundred:=maxpowerpoint/100 MOD 10;
//str:=CONCAT(str,UDINT_TO_STRING(_hundred));
//_ten:=maxpowerpoint/10 MOD 10;
//str:=CONCAT(str,UDINT_TO_STRING(_ten));
//_bit:=maxpowerpoint MOD 10;
//str:=CONCAT(str,UDINT_TO_STRING(_bit));
str:=CONCAT(str,' M$R');
appendSend(str);
END_METHOD

METHOD WritePower : BOOL
VAR_INPUT
	powerpoint:UDINT;
END_VAR
VAR
	str:STRING;
	_bit:UDINT;
	_ten:UDINT;
	_hundred:UDINT;
	_thousand:UDINT;
END_VAR
str:='';
//_thousand:=powerpoint/1000;
str:=CONCAT(str,UDINT_TO_STRING(powerpoint));
//_hundred:=powerpoint/100 MOD 10;
//str:=CONCAT(str,UDINT_TO_STRING(_hundred));
//_ten:=powerpoint/10 MOD 10;
//str:=CONCAT(str,UDINT_TO_STRING(_ten));
//_bit:=powerpoint MOD 10;
//str:=CONCAT(str,UDINT_TO_STRING(_bit));
str:=CONCAT(str,' W$R');
appendSend(str);
END_METHOD

METHOD WriteReset : BOOL
VAR_INPUT
		

END_VAR
appendSend('RESET$R');
END_METHOD

METHOD WriteRS232Mode : BOOL
VAR_INPUT
		

END_VAR
appendSend('***$R');
END_METHOD

METHOD WriteStart : BOOL
VAR_INPUT
		

END_VAR
appendSend('G$R');
END_METHOD

METHOD WriteStop : BOOL
VAR_INPUT
		

END_VAR
appendSend('S$R');
END_METHOD

END_PROGRAM

// ---- POUs/BaseModule/Error/error_Printf.TcPOU
//设备报警信息打印
FUNCTION error_Printf : BOOL
VAR_INPUT
	errorID					:DINT;
END_VAR
VAR
	sErrTXT					:STRING(255);
	sErrWTXT				:WSTRING(255);
END_VAR

sErrTXT:=errorMonitor.getErrTXT(errorID);
sErrWTXT:=errorMonitor.getErrWTXT(errorID);
IF gCNErrShow THEN
	gLog.append_EX(sErrWTXT);
	gErrWTxtShow:=sErrWTXT;
ELSE
	gLog.append(sErrTXT);
	gErrTxtShow:=sErrTXT;
	gErrWTxtShow:=TO_WSTRING(gErrTxtShow);
END_IF

END_FUNCTION

// ---- POUs/BaseModule/DataSaveModule_EX/RecipeNameModule_EX.TcPOU
FUNCTION_BLOCK RecipeNameModule_EX
VAR_INPUT
	sFileName						:T_MaxString:='C:\GideonSaveData.csv';//'Hard Disk\IASaveData.csv'  数据文件存储路径
	readB							:BOOL:=FALSE;//读取触发
	saveB							:BOOL:=FALSE;//保存触发
	deleteB							:BOOL:=FALSE;// 删除触发
	dataString						:ARRAY[0..gRecipeNameMAX_CSV_ROWS, 0..gRecipeNameMAX_CSV_COLUMNS ] OF STRING(30);
	pDatabaseHMI					:ARRAY[1..gRecipeNameMAX_CSV_ROWS+1] OF RecipeNamePar;(* Target PLC database *)
	pDatabase						:ARRAY[0..gRecipeNameMAX_CSV_ROWS, 0..gRecipeNameMAX_CSV_COLUMNS ] OF STRING(30);(* Target PLC database *)
	dataStringLength				:UDINT:=99;
END_VAR
VAR_OUTPUT
	busy							:BOOL:=FALSE;
	rDone							:BOOL:=FALSE;
	sDone							:BOOL:=FALSE;
	error							:BOOL:=FALSE;
	errID							:UDINT:=0;
	errTxt							:STRING(255):='';
	outData							:ARRAY [1..gRecipeNameMAX_String_NUM] OF RecipeNamePar; 
END_VAR
VAR_IN_OUT
	
END_VAR
VAR	
	csv_rows						:UDINT:=gRecipeNameMAX_CSV_ROWS;
	csv_columns						:UDINT:=gRecipeNameMAX_CSV_COLUMNS;
	startUpB						:BOOL:=FALSE;
	writeTxt						:P_TextModeWrite_RecipeName;
	readTxt							:P_TextModeRead_RecipeName;
	deleteTxt						:P_TextModeDelete_1;
	fbFileOpen						:FB_FileOpen;//检查文件是否存在
	fbFileClose						:FB_FileClose;(* Closes file *)
	hFile							:UINT:=0;(* File handle of the source file *)
	checkFileExistError				:BOOL;
	initB							:BOOL:=FALSE;
	saveStep						:UINT:=0;
	deleteStep						:UINT:=0;
	readStep						:UINT:=0;
	sFileNameOld					:T_MaxString;//旧文件名
//获取系统时间
	ntGetTime				: NT_GetTime;
	systemTimeStruct		: TIMESTRUCT;
	getSystemTimeStep		: UINT:=0;
	systemTIMEStr			: STRING:='';//系统时间，格式YYYY-MM-DD hh:mm:ss_zzz
	systemTIMEStr2			: STRING:='';//系统时间，格式YYYYMMDDhhmmss
	sysTIMEStrYY			: STRING:='';//系统时间，年
	sysTIMEStrMM			: STRING:='';//系统时间，月
	sysTIMEStrDD			: STRING:='';//系统时间，日
	sysTIMEStr_HH			: STRING:='';//系统时间，时
	sysTIMEStr_mm			: STRING:='';//系统时间，分
	sysTIMEStr_ss			: STRING:='';//系统时间，秒
END_VAR

IF dataStringLength>gRecipeNameMAX_String_NUM THEN
	dataStringLength:=gRecipeNameMAX_String_NUM;
END_IF


csv_rows:=dataStringLength + 1;
IF csv_rows>gRecipeNameMAX_CSV_ROWS THEN
	csv_rows:=gRecipeNameMAX_CSV_ROWS;
END_IF

//judge length
IF gRecipeNameMAX_CSV_ROWS<(dataStringLength+1) THEN
	error:=TRUE;
	errTxt:='dataBase$'s length too short';
	RETURN;
END_IF
IF csv_rows<(dataStringLength+1) THEN
	error:=TRUE;
	errTxt:='dataBase$'s length too short';
	RETURN;
END_IF

init();
IF initB THEN
	readMethod();
	saveMethod();
END_IF
getSystemTime();

METHOD PRIVATE createDir : BOOL
VAR
	sPathNameTemp	: T_MaxString := 'C:\TwinCAT\Data.txt';
	sDriveTemp		: STRING(3);
	sDirTemp		: T_MaxString;
	sFileNameTemp	: T_MaxString;
	sExtTemp		: T_MaxString;
	bSuccess		: BOOL;
	fbCreateDir		: FB_CreateDir;
	fbCreateDir2	: FB_CreateDir;
	sFileDirTemp	: T_MaxString;
	sFileDirTemp2	: T_MaxString;
END_VAR
sPathNameTemp:=sFileName;
bSuccess := F_SplitPathName( sPathName := sPathNameTemp,
	sDrive := sDriveTemp,
	sDir := sDirTemp,
	sFileName := sFileNameTemp,
	sExt := sExtTemp );
IF bSuccess THEN
	bSuccess:=FALSE;
	IF LEFT(sDirTemp,LEN(sDirTemp)-1) <> '' THEN
		//sFileDirTemp:=CONCAT(STR1:=sDriveTemp,STR2:=LEFT(sDirTemp,LEN(sDirTemp)-1));
		//sFileNameOld:=CONCAT(STR1:=sFileDirTemp,STR2:=CONCAT('\',CONCAT(sFileNameTemp,'_Old.csv')));//用于重命名参数文件
		sFileDirTemp:='';
		sFileDirTemp:=CONCAT(sFileDirTemp,sDriveTemp);
		sFileDirTemp:=CONCAT(sFileDirTemp,LEFT(sDirTemp,LEN(sDirTemp)-1));
		sFileDirTemp2:='';
		sFileDirTemp2:=CONCAT(sFileDirTemp2,sFileDirTemp);
		sFileDirTemp2:=CONCAT(sFileDirTemp2,'\Old');
		
		sFileNameOld:='';
		sFileNameOld:=CONCAT(sFileNameOld,sFileDirTemp);
		sFileNameOld:=CONCAT(sFileNameOld,'\Old\');//'\'
		sFileNameOld:=CONCAT(sFileNameOld,sFileNameTemp);
		sFileNameOld:=CONCAT(sFileNameOld,'_Old_');
		sFileNameOld:=CONCAT(sFileNameOld,systemTIMEStr2);
		sFileNameOld:=CONCAT(sFileNameOld,'.csv');
		
		fbCreateDir(
			sNetId:= , 
			sPathName:= sFileDirTemp, 
			ePath:= PATH_GENERIC, 
			bExecute:= TRUE, 
			tTimeout:= , 
			bBusy=> , 
			bError=> , 
			nErrId=> );
		fbCreateDir2(
			sNetId:= , 
			sPathName:= sFileDirTemp2, 
			ePath:= PATH_GENERIC, 
			bExecute:= TRUE, 
			tTimeout:= , 
			bBusy=> , 
			bError=> , 
			nErrId=> );
	END_IF
END_IF
fbCreateDir(
	sNetId:= , 
	sPathName:= , 
	ePath:= , 
	bExecute:= FALSE, 
	tTimeout:= , 
	bBusy=> , 
	bError=> , 
	nErrId=> );
fbCreateDir2(
	sNetId:= , 
	sPathName:= , 
	ePath:= , 
	bExecute:= FALSE, 
	tTimeout:= , 
	bBusy=> , 
	bError=> , 
	nErrId=> );
END_METHOD

METHOD PRIVATE data2String : BOOL
VAR_INPUT
END_VAR
VAR
	i:UDINT:=0;
END_VAR
//judge length
IF gRecipeNameMAX_CSV_ROWS<(gRecipeNameMAX_String_NUM+1) THEN
	error:=TRUE;
	errTxt:='dataBase$'s length too short';
	RETURN;
END_IF
IF csv_rows<(dataStringLength+1) THEN
	error:=TRUE;
	errTxt:='dataBase$'s length too short';
	RETURN;
END_IF


//bool
FOR i:=0 TO dataStringLength DO
	pDatabase[i+1,0]:=TO_STRING(i);//num
	pDatabase[i+1,1]:=gRecipeNameSelect[i+1].Name;//Name
	pDatabase[i+1,2]:='1';;//ID
	pDatabase[i+1,3]:='Null';//Par1
	pDatabase[i+1,4]:='Null';//Par2
END_FOR
END_METHOD

METHOD PRIVATE deleteMethod : BOOL
VAR_INPUT
END_VAR
CASE deleteStep OF
0:
	IF deleteB AND (NOT busy) THEN
		deleteStep:=1;
		deleteB:=FALSE;
		busy:=TRUE;
		sDone:=FALSE;
		error:=FALSE;
		errID:=0;
		errTxt:='';
	END_IF

1:
	deleteStep:=2;

2:
	deleteTxt(
	bDelete:=TRUE , 
	sFileName:=sFileName , 
	sFileNameOld:= , 
	bBusy=> , 
	error=> , 
	nErrId=> );	
	deleteStep:=3;

3:
	deleteTxt.bDelete:=FALSE;
	
	IF error THEN
		deleteStep:=110;
		RETURN;
	END_IF

	IF NOT writeTxt.bBusy THEN
		deleteStep:=100;
	END_IF

100:
	busy:=FALSE;
	sDone:=TRUE;
	error:=error;
	errID:=errID;
	errTxt:=errTxt;

	IF NOT deleteB THEN
		deleteStep:=0;
	END_IF

110:
	busy:=FALSE;
	sDone:=FALSE;
	error:=TRUE;
	errID:=errID;
	errTxt:='save data fail';

	IF NOT deleteB THEN
		deleteStep:=0;
	END_IF
END_CASE
deleteTxt(
	bDelete:= , 
	sFileName:=sFileName , 
	sFileNameOld:= , 
	bBusy=> , 
	error=> , 
	nErrId=> );
END_METHOD

METHOD deleteSlector : BOOL
VAR_INPUT
	recipeSelect					:ARRAY [1..10] OF STRING;
	inidex							:INT;
END_VAR
VAR_OUTPUT
	error:BOOL;
	outrecipeSelect					:ARRAY [1..10] OF STRING;
END_VAR
VAR
	itemp:INT;
END_VAR
outrecipeSelect:=recipeSelect;
IF inidex>0 AND inidex<=gRecipeSelctMaxIndex THEN
	FOR itemp:=inidex TO gRecipeSelctMaxIndex-1 BY 1 DO
		outrecipeSelect[itemp]:=outrecipeSelect[itemp+1];
	END_FOR
	outrecipeSelect[gRecipeSelctMaxIndex]:='';
	error:=FALSE;
ELSE
	error:=TRUE;
END_IF
END_METHOD

METHOD PRIVATE getSystemTime : BOOL
VAR_INPUT
END_VAR
//获取本地系统时间--输出到变量 systemTIMEStr
CASE getSystemTimeStep OF
0:
	ntGetTime(
		NETID:= , 
		START:= FALSE, 
		TMOUT:= , 
		BUSY=> , 
		ERR=> , 
		ERRID=> , 
		TIMESTR=> systemTimeStruct);
	IF NOT ntGetTime.BUSY AND NOT ntGetTime.ERR THEN
		getSystemTimeStep:=getSystemTimeStep+1;
	END_IF
1:
	ntGetTime(
		NETID:= , 
		START:= TRUE, 
		TMOUT:= , 
		BUSY=> , 
		ERR=> , 
		ERRID=> , 
		TIMESTR=> systemTimeStruct);
	IF NOT ntGetTime.BUSY AND NOT ntGetTime.ERR THEN
		systemTIMEStr:=SYSTEMTIME_TO_STRING(systemTimeStruct);//系统时间转成字符串格式
		
		sysTIMEStrYY:=WORD_TO_DECSTR(in:=systemTimeStruct.wYear,iPrecision:=4);
		sysTIMEStrMM:=WORD_TO_DECSTR(in:=systemTimeStruct.wMonth,iPrecision:=2);
		sysTIMEStrDD:=WORD_TO_DECSTR(in:=systemTimeStruct.wDay,iPrecision:=2);
		sysTIMEStr_HH:=WORD_TO_DECSTR(in:=systemTimeStruct.wHour,iPrecision:=2);
		sysTIMEStr_mm:=WORD_TO_DECSTR(in:=systemTimeStruct.wMinute,iPrecision:=2);
		sysTIMEStr_ss:=WORD_TO_DECSTR(in:=systemTimeStruct.wSecond,iPrecision:=2);
		
		systemTIMEStr2:='';
		systemTIMEStr2:=CONCAT(systemTIMEStr2,sysTIMEStrYY);
		systemTIMEStr2:=CONCAT(systemTIMEStr2,sysTIMEStrMM);
		systemTIMEStr2:=CONCAT(systemTIMEStr2,sysTIMEStrDD);
		systemTIMEStr2:=CONCAT(systemTIMEStr2,sysTIMEStr_HH);
		systemTIMEStr2:=CONCAT(systemTIMEStr2,sysTIMEStr_mm);
		systemTIMEStr2:=CONCAT(systemTIMEStr2,sysTIMEStr_ss);
		
		getSystemTimeStep:=0;
	ELSIF ntGetTime.ERR THEN
		systemTIMEStr:='';
		getSystemTimeStep:=0;
	END_IF	
END_CASE
END_METHOD

METHOD getValue : BOOL
VAR_IN_OUT
	value:STRING;
END_VAR
VAR_INPUT
	cnum:UDINT;
	rnum:UDINT;
END_VAR
IF 0<=rnum AND rnum<=dataStringLength
	AND 0<=cnum AND cnum<=gRecipeMAX_CSV_COLUMNS THEN
	value:=pDatabase[rnum,cnum];
	getValue:=TRUE;
ELSE
	value:='';
	getValue:=FALSE;
END_IF
END_METHOD

METHOD PRIVATE init : BOOL
VAR_INPUT
END_VAR
VAR
	i:UDINT:=0;
END_VAR
//创建生成初始表格
//judge length
IF gRecipeNameMAX_CSV_ROWS<(gRecipeNameMAX_String_NUM+1) THEN
	error:=TRUE;
	errTxt:='dataBase$'s length too short';
	RETURN;
END_IF
IF csv_rows<(dataStringLength+1) THEN
	error:=TRUE;
	errTxt:='dataBase$'s length too short';
	RETURN;
END_IF


IF initB AND (NOT busy) THEN
	RETURN;
END_IF
initB:=TRUE;

//header
	pDatabase[0,0]:='NUM';//NUM
	pDatabase[0,1]:='RecipeName';//Name
	pDatabase[0,2]:='RecipeID';//ID
	pDatabase[0,3]:='Par1';//Par1
	pDatabase[0,4]:='Par2';//Par2
	
(*--- 不在此处填充，转移到保存数据时填充
//bool
FOR i:=1 TO (dataBoolLength+1) DO
	//pDatabase[i,0]:=UDINT_TO_STRING(i-1);//NUM  --- 不在此处填充
	//pDatabase[i,1]:='BOOL';//data type --- 不在此处填充
	//pDatabase[i,2]:='';//name
	//pDatabase[i,3]:=BOOL_TO_STRING(FALSE);//value
	//pDatabase[i,4]:='';//no use
END_FOR

//dint
FOR i:=(dataBoolLength+2) TO (dataBoolLength+2+dataDintLength) DO
	//pDatabase[i,0]:=UDINT_TO_STRING(i-(dataBoolLength+2));//NUM  --- 不在此处填充
	//pDatabase[i,1]:='DINT';//data type --- 不在此处填充
	//pDatabase[i,2]:='';//name
	//pDatabase[i,3]:=DINT_TO_STRING(0);//value
	//pDatabase[i,4]:='';//no use
END_FOR

//lreal
FOR i:=(dataBoolLength+dataDintLength+3) TO (dataBoolLength+dataDintLength+dataLrealLength+3) DO
	//pDatabase[i,0]:=UDINT_TO_STRING(i-(dataBoolLength+dataDintLength+3));//NUM  --- 不在此处填充
	//pDatabase[i,1]:='LREAL';//data type --- 不在此处填充
	//pDatabase[i,2]:='';//name
	//pDatabase[i,3]:=DINT_TO_STRING(0);//value
	//pDatabase[i,4]:='';//no use
END_FOR
*)
END_METHOD

METHOD PRIVATE readMethod : BOOL
VAR_INPUT
END_VAR
CASE readStep OF
0:
	IF (readB OR (NOT startUPb)) AND (NOT busy) THEN
		readStep:=1;
		startUPb:=TRUE;//for first time, 
		readB:=FALSE;
		rDone:=FALSE;
		busy:=TRUE;
		error:=FALSE;
		errID:=0;
		errTxt:='';
		fbFileOpen(bExecute:= FALSE);
		checkFileExistError:=FALSE;
	END_IF
	
1:
	fbFileOpen(
		sNetId:= , 
		sPathName:= sFileName, 
		nMode:= FOPEN_MODEREAD, 
		ePath:= PATH_GENERIC, 
		bExecute:= TRUE, 
		tTimeout:= , 
		bBusy=> , 
		bError=> , 
		nErrId=> , 
		hFile=> hFile);
	IF NOT fbFileOpen.bBusy THEN
		IF fbFileOpen.bError THEN
			checkFileExistError:=TRUE;
		END_IF
		fbFileOpen(bExecute:= FALSE);
		readStep:=2;
	END_IF
	fbFileClose(bExecute:= FALSE);
2:
	fbFileClose(
		sNetId:= , 
		hFile:= hFile, 
		bExecute:= TRUE, 
		tTimeout:= , 
		bBusy=> , 
		bError=> , 
		nErrId=> );
	IF NOT fbFileClose.bBusy THEN
		IF checkFileExistError THEN
			readStep:=110;
		ELSE
			readStep:=11;
		END_IF
		fbFileClose(bExecute:= FALSE);
	END_IF

11:
	//read txt to Database
	readTxt(
		database:= pDatabase, 
		csv_rows:= csv_rows, 
		csv_columns:= csv_columns, 
		bRead:= TRUE, 
		sFileName:= sFileName);
	readStep:=12;

12:
	readTxt(
		database:= pDatabase, 
		csv_rows:= csv_rows, 
		csv_columns:= csv_columns, 
		bRead:= FALSE, 
		sFileName:= sFileName,
		Error=>error,
		nErrId=>errID);
		
	IF error THEN
		readStep:=110;
		RETURN;
	END_IF
	
	IF NOT readTxt.bBusy THEN
		readStep:=13;
	END_IF
	
13:
	string2Data();
	readStep:=100;
	
100:
	rDone:=TRUE;
	busy:=FALSE;
	error:=error;
	errID:=errID;
	errTxt:=errTxt;
	IF NOT readB THEN
		readStep:=0;
	END_IF	


110:
	rDone:=FALSE;
	busy:=FALSE;
	error:=TRUE;
	errID:=errID;
	errTxt:='read data fail';	
	IF NOT readB THEN
		readStep:=0;
	END_IF		
	gRecipeSelectIndex1:=1;
END_CASE
END_METHOD

METHOD PRIVATE saveMethod : BOOL
VAR_INPUT
END_VAR
CASE saveStep OF
0:
	IF saveB AND (NOT busy) THEN
		saveStep:=1;
		saveB:=FALSE;
		busy:=TRUE;
		sDone:=FALSE;
		error:=FALSE;
		errID:=0;
		errTxt:='';
	END_IF

1:
	createDir();
	data2String();
	saveStep:=2;

2:
	writeTxt(
		database:= pDatabase, 
		csv_rows:= csv_rows, 
		csv_columns:= csv_columns, 
		bWrite:= TRUE, 
		sFileName:= sFileName,
		sFileNameOld:= sFileNameOld);	
	saveStep:=3;

3:
	writeTxt(
		database:= pDatabase, 
		csv_rows:= csv_rows, 
		csv_columns:= csv_columns, 
		bWrite:= FALSE, 
		sFileName:= sFileName,
		sFileNameOld:= sFileNameOld,
		Error=>error,
		nErrID=>errID);	
	
	IF error THEN
		saveStep:=110;
		RETURN;
	END_IF

	IF NOT writeTxt.bBusy THEN
		saveStep:=100;
	END_IF

100:
	busy:=FALSE;
	sDone:=TRUE;
	error:=error;
	errID:=errID;
	errTxt:=errTxt;

	IF NOT saveB THEN
		saveStep:=0;
	END_IF

110:
	busy:=FALSE;
	sDone:=FALSE;
	error:=TRUE;
	errID:=errID;
	errTxt:='save data fail';

	IF NOT saveB THEN
		saveStep:=0;
	END_IF
END_CASE
END_METHOD

METHOD setValue : BOOL
VAR_INPUT
	value:STRING;
END_VAR
VAR_INPUT
	rnum:UDINT;
	cnum:UDINT;
END_VAR
IF 0<=rnum AND rnum<=dataStringLength
	AND 0<=cnum AND cnum<=gRecipeMAX_CSV_COLUMNS THEN
	pDatabase[rnum,cnum]:=value;
	setValue:=TRUE;
ELSE
	setValue:=FALSE;
END_IF
END_METHOD

METHOD PRIVATE string2Data : BOOL
VAR_INPUT
END_VAR
VAR
	i:INT:=0;
	index_temp:UDINT;
END_VAR
//judge length
IF gRecipeNameMAX_CSV_ROWS<(gRecipeNameMAX_String_NUM+1) THEN
	error:=TRUE;
	errTxt:='dataBase$'s length too short';
	RETURN;
END_IF
IF csv_rows<(dataStringLength+1) THEN
	error:=TRUE;
	errTxt:='dataBase$'s length too short';
	RETURN;
END_IF

(*
//bool
FOR i:=0 TO dataBoolLength DO
	dataBool[i]:=STRING_TO_BOOL(pDatabase[i+1,3]);//value
END_FOR

//dint
FOR i:=(dataBoolLength+1) TO (dataBoolLength+1+dataDintLength) DO
	dataDint[i-(dataBoolLength+1)]:=STRING_TO_DINT(pDatabase[i+1,3]);//value
END_FOR

//lreal
FOR i:=(dataBoolLength+dataDintLength+2) TO (dataBoolLength+dataDintLength+dataLrealLength+2) DO
	dataLreal[i-(dataBoolLength+dataDintLength+2)]:=STRING_TO_LREAL(pDatabase[i+1,3]);//value
END_FOR
*)
FOR i:=0 TO UDINT_TO_INT(gRecipeNameMAX_CSV_ROWS)  DO
	dataString[i,0]:=(pDatabase[i,0]);
	dataString[i,1]:=(pDatabase[i,1]);
	dataString[i,2]:=(pDatabase[i,2]);
	dataString[i,3]:=(pDatabase[i,3]);
	dataString[i,4]:=(pDatabase[i,4]);
	
	
	IF i<UDINT_TO_INT(gRecipeNameMAX_CSV_ROWS) THEN
		gRecipeSelectStruct[i+1].NUM:=(pDatabase[i+1,0]);
		gRecipeSelectStruct[i+1].Name:=(pDatabase[i+1,1]);
		gRecipeSelectStruct[i+1].ID:=(pDatabase[i+1,2]);
		gRecipeSelectStruct[i+1].Note1:=(pDatabase[i+1,3]);
		gRecipeSelectStruct[i+1].Note2:=(pDatabase[i+1,4]);
		
		gRecipeNameSelect[i+1].Name:=gRecipeSelectStruct[i+1].Name;
		
		IF len(gRecipeSelectStruct[i+1].Name)>0 THEN
			gRecipeNameMax:=INT_TO_UDINT(i)+1;
		END_IF
	END_IF
END_FOR

FOR  i:=1 TO gRecipeSelctMaxIndex DO
	gRecipeNameSelectShow[i]:=gRecipeNameSelect[i];
END_FOR
END_METHOD

ACTION VersionLog:
(*
版本: V1.0.0.0 20241012  CPH
说明:
	1. 首个版本
(**************************************************)
版本: V1.0.0.1
说明:
	1. 增加参数备份文件，文件名以原文件名+时间命名
(**************************************************)
*)
END_ACTION

END_FUNCTION_BLOCK

// ---- POUs/BaseModule/DataSaveModule_EX/csvReadWriteInTextMode/P_TextModeWrite_RecipeName.TcPOU
FUNCTION_BLOCK P_TextModeWrite_RecipeName
VAR_IN_OUT
	database		: ARRAY[0..gRecipeNameMAX_CSV_ROWS, 0..gRecipeNameMAX_CSV_COLUMNS ] OF STRING(30);
	csv_rows		: UDINT;
	csv_columns		: UDINT;
END_VAR
VAR_INPUT
	bWrite			: BOOL := FALSE;(* Rising edge starts program execution *)	
	sFileName		: T_MaxString := '';(* CSV destination file path and name *)
	sFileNameOld	:T_MaxString := '';(*旧文件名*)
END_VAR
VAR_OUTPUT
	bBusy			: BOOL;
	error			: BOOL;
	nErrId			: UDINT;	
END_VAR
VAR
	bError			: BOOL;
	sNetId			: T_AmsNetId := '';	(* TwinCAT system network address *)

	sCSVLine		: T_MaxString := '';(* Single CSV text line (row, record), we are using string as record buffer (your are able to see created fields) *)
	sCSVField		: T_MaxString := '';(* Single CSV field value (column, record field) *)
	//sCSVField		: UDINT;

	nRow	 		: UDINT 	:= 0;(* Row number (record) *)
	nColumn			: UDINT 	:= 0;(* Column number (record field) *)
	hFile			: UINT		:= 0;(* File handle of the source file *)
	step			: DWORD 	:= 0;
	fbFileOpen		: FB_FileOpen;(* Opens file *)
	fbFileClose		: FB_FileClose;(* Closes file *)
	fbFilePuts		: FB_FilePuts;(* Writes one record (line) *)
	fbFileWrite     : FB_FileWrite;
	fbWriter		: FB_CSVMemBufferWriter;(* Helper function block used to create CSV data bytes (single record line) *)
    StringModelWrite		: StringModel_256000_EX;
	fbFileRename			: FB_FileRename;//修改文件名称
	fbFileDelete			: FB_FileDelete;//删除文件
	writeTON				: TON;//延时写入

	(* :=[ (* Source PLC database *)
	'0_0', '0_1', '0_2', '0_3', '0_4', '0_5',
	'1_0', '1_1', '1_2', '1_3', '1_4', '1_5',
	'2_0', '2_1', '2_2', '2_3', '2_4', '2_5',
	'3_0', '3_1', '3_2', '3_3', '3_4', '3_5',
	'4_0', '4_1', '4_2', '4_3', '4_4', '4_5',
	'5_0', '5_1', '5_2', '5_3', '5_4', '5_5'];*)

END_VAR

DEFAULT_CSV_FIELD_SEP:= 16#2C;  //配置CSV文件的分割符，16#2C表明各个参数之间是用逗号分隔的。
CASE step OF
	0:(* Wait for rising edge at bWrite variable *)
		IF bWrite THEN
			bWrite 	:= FALSE;
			bBusy 	:= TRUE;
			error	:= FALSE;
			bError	:= FALSE;
			nErrId	:= 0;
			hFile	:= 0;
			nRow	:= 0;
			nColumn	:= 0;
			step 	:= 1;
		END_IF
	1:
		StringModelWrite.init();
		fbFileDelete(bExecute:= FALSE);
		fbFileRename(bExecute:= FALSE);
		step:=2;
	2:
		fbFileDelete(
			sNetId:= , 
			sPathName:= sFileNameOld, 
			ePath:= PATH_GENERIC, 
			bExecute:= TRUE, 
			tTimeout:= DEFAULT_ADS_TIMEOUT, 
			bBusy=> , 
			bError=> , 
			nErrId=> );
		step:=3;
	3:
		fbFileDelete(bExecute:= FALSE);
		IF NOT fbFileDelete.bBusy THEN
			step:=4;
		END_IF
	4:
		fbFileRename(
			sNetId:= , 
			sOldName:= sFileName, 
			sNewName:= sFileNameOld, 
			ePath:= PATH_GENERIC, 
			bExecute:= TRUE, 
			tTimeout:= DEFAULT_ADS_TIMEOUT, 
			bBusy=> , 
			bError=> , 
			nErrId=> );
		step:=5;
	5:
		fbFileRename(bExecute:= FALSE);
		IF NOT fbFileRename.bBusy THEN
			step:=10;
		END_IF

	10:(* Open source file *)
		fbFileOpen(  bExecute := FALSE  );
		fbFileOpen( sNetId := sNetId, sPathName := sFileName, nMode := FOPEN_MODEWRITE OR FOPEN_MODETEXT,(* Open file in TEXT mode! *)
					ePath := PATH_GENERIC, bExecute := TRUE );
		step := 20;

	20:(* Wait until open not busy *)
		//StringModelWrite.init();
		fbFileOpen( bExecute := FALSE, bError => bError, nErrID => nErrID, hFile => hFile );
		IF NOT fbFileOpen.bBusy THEN
			IF NOT fbFileOpen.bError THEN
				step := 30;
			ELSE(* Error: file not found? *)
				step := 1000;
			END_IF
		END_IF
	
	30:(* Convert one PLC record to CSV format *)
		FOR nRow:=0 TO csv_rows BY 1 DO
				sCSVLine := '';
				fbWriter.eCmd := eEnumCmd_First;(* Write first field value *)
			FOR nColumn := 0 TO csv_columns BY 1 DO
				sCSVField := STRING_TO_CSVFIELD( database[ nRow, nColumn ], FALSE );(* TODO: Get field value from your application *)
				(* Add new field to the record buffer *)
				fbWriter( 	pBuffer := ADR( sCSVLine ), cbBuffer := SIZEOF( sCSVLine ) - 1, putValue := sCSVField, pValue := 0, cbValue := 0,
							bCRLF := ( nColumn = csv_columns ) );(* bCRLF == TRUE => Write CRLF after the last field value *)
				IF fbWriter.bOk THEN
					fbWriter.eCmd := eEnumCmd_Next;(* Write next field value *)
				ELSE(* Error *)
					step := 1000;
					RETURN;
				END_IF
			END_FOR
			(* FB_FilePuts adds allready CR (carriage return) to the written line.
			We have to replace the $R$L characters with $L character to avoid double CR. *)
			IF RIGHT( sCSVLine, 2 ) = '$R$L' THEN
				sCSVLine := REPLACE( sCSVLine, '$L', 2, LEN( sCSVLine ) - 1 );
			END_IF
            StringModelWrite.append(str:= sCSVLine);
		END_FOR
		IF nRow> csv_rows THEN
			step := 40;(* Write record to the file *)
		END_IF
		writeTON(IN:=FALSE);

	40:(* Write record to file *)
		fbFileWrite( bExecute := FALSE );
		writeTON(IN:=NOT writeTON.Q,PT:=T#50MS);
		IF writeTON.Q THEN
			//fbFileWrite( sNetId := sNetId, hFile := hFile, pWriteBuff := StringModelWrite.getAddr, cbWriteLen := StringModelWrite.length, bExecute := TRUE );
			fbFileWrite( sNetId := sNetId, hFile := hFile, pWriteBuff := ADR(StringModelWrite.b), cbWriteLen := StringModelWrite.length, bExecute := TRUE );
			step := 50;
		END_IF

	50:(* Wait until write not busy *)
		fbFileWrite( bExecute := FALSE, bError => bError, nErrID => nErrID );
		IF NOT fbFileWrite.bBusy THEN
			IF NOT fbFileWrite.bError THEN
				step := 100;(* Write next record *)
			ELSE(* Error *)
				step := 1000;
			END_IF
		END_IF
		
	100:(* Close source file *)
		fbFileClose( bExecute := FALSE );
		fbFileClose( sNetId := sNetId, hFile := hFile, bExecute := TRUE );
		step := 110;

	110:(* Wait until close not busy *)
		fbFileClose( bExecute := FALSE, bError => bError, nErrID => nErrID );
		IF NOT fbFileClose.bBusy THEN
			hFile := 0;
			step := 1000;
		END_IF

	1000:(* Error or ready step => cleanup *)
		IF ( hFile <> 0 ) THEN
			step := 100; (* Close the source file *)
		ELSE
			bBusy := FALSE;
			error := bError;
			step := 0;	(* Ready *)
		END_IF
END_CASE

END_FUNCTION_BLOCK

// ---- POUs/BaseModule/DataSaveModule_EX/csvReadWriteInTextMode/P_TextModeRead_RecipeName.TcPOU
FUNCTION_BLOCK P_TextModeRead_RecipeName
VAR_IN_OUT
	database		: ARRAY[0..gRecipeNameMAX_CSV_ROWS, 0..gRecipeNameMAX_CSV_COLUMNS ] OF STRING(30);(* Target PLC database *)
	csv_rows		: UDINT;
	csv_columns		: UDINT;
END_VAR
VAR_INPUT
	bRead			: BOOL := FALSE;(* Rising edge starts program execution *)	
	sFileName		: T_MaxString := '';(* CSV source file path and name *)
END_VAR
VAR_OUTPUT
	bBusy			: BOOL;
	error			: BOOL;
	nErrId			: UDINT;	
END_VAR
VAR
	bError			: BOOL;
	sNetId			: T_AmsNetId := '';	(* TwinCAT system network address *)
	sCSVLine		: T_MaxString := '';(* Single CSV text line (row, record), we are using string as record buffer (your are able to see read fields)  *)
	sCSVField		: T_MaxString := '';(* Single CSV field value (column, record field) *)
	nRow	 		: UDINT 	:= 0;(* Row number (record) *)
	nColumn			: UDINT 	:= 0;(* Column number (record field) *)
	hFile			: UINT		:= 0;(* File handle of the source file *)
	step			: DWORD 	:= 0;
	fbFileOpen		: FB_FileOpen;(* Opens file *)
	fbFileClose		: FB_FileClose;(* Closes file *)
	fbFileGets		: FB_FileGets;(* Reads one record (line) *)
	fbFileRead		: FB_FileRead;//---------------------------------------
	fbReader		: FB_CSVMemBufferReader;(* Helper function block used to parse CSV data bytes (single record line) *)
	
	readData:ARRAY[gNumBegin..(gMaxNumLength+gNumBegin-1)]OF BYTE;
	strTemp : T_MaxString;
	strT : T_MaxString;
	i : UDINT:=0;
	iTemp : UDINT:=0;
END_VAR

DEFAULT_CSV_FIELD_SEP:= 16#2C;  //配置CSV文件的分割符，16#2C表明各个参数之间是用逗号分隔的。
CASE step OF
	0:	(* Wait for rising edge at bRead variable *)
		IF bRead THEN
			bRead 	:= FALSE;
			bBusy 	:= TRUE;
			error:= bError	:= FALSE;
			nErrId	:= 0;
			hFile	:= 0;
			nRow	:= 0;
			nColumn	:= 0;
			MEMSET( ADR( database ), 0, SIZEOF( database ) );
			step 		:= 1;
		END_IF

	1:	(* Open source file *)
		fbFileOpen(  bExecute := FALSE  );
		fbFileOpen( sNetId := sNetId, sPathName := sFileName, nMode := FOPEN_MODEREAD OR FOPEN_MODETEXT,(* Open file in TEXT mode! *)
					ePath := PATH_GENERIC, bExecute := TRUE );
		step := 2;

	2:(* Wait until open not busy *)
		fbFileOpen( bExecute := FALSE, bError => bError, nErrID => nErrID, hFile => hFile );
		IF NOT fbFileOpen.bBusy THEN
			IF NOT fbFileOpen.bError THEN
				step := 3;
			ELSE(* Error: file not found? *)
				step := 100;
			END_IF
		END_IF
		
	3:
		step := 4;
	4:
		fbFileRead(
			sNetId:= sNetId, 
			hFile:= hFile, 
			bExecute:= FALSE,);
		step := 5;
	5:(*Read data from file*)
		fbFileRead(
			sNetId:= sNetId, 
			hFile:= hFile, 
			pReadBuff:= ADR(readData),
			cbReadLen:= gMaxNumLength,
			bExecute:= TRUE, 
			tTimeout:= , 
			bBusy=> , 
			bError=> , 
			nErrId=> , 
			cbRead=> , 
			bEOF=> );
		IF NOT fbFileRead.bBusy AND NOT fbFileRead.bError THEN
			IF fbFileRead.bEOF THEN
				step := 6;
			END_IF
			step := 6;
			fbFileRead(
				sNetId:= sNetId, 
				hFile:= hFile, 
				bExecute:= FALSE,);
		ELSIF fbFileRead.bError THEN
			step := 100;
		END_IF
		sCSVLine := '';
		iTemp:=1;
	6:
		FOR nRow:=0 TO csv_rows BY 1 DO
			sCSVLine := '';
			FOR i:=iTemp TO gMaxNumLength BY 1 DO
				strT := F_ToCHR(c:=readData[i]);
				IF '$L' = strT THEN
					strTemp:=CONCAT(STR1:=sCSVLine,STR2:='$R$L');
					iTemp:=i+1;
					EXIT;
				ELSE
					sCSVLine:=CONCAT(STR1:=sCSVLine,STR2:=strT);
				END_IF
			END_FOR
			fbReader.eCmd := eEnumCmd_First;(* Read first field value *)
			FOR nColumn := 0 TO csv_columns BY 1 DO
				fbReader( pBuffer := ADR( sCSVLine ), cbBuffer := SIZEOF( sCSVLine ), getValue => sCSVField);
				IF fbReader.bOk THEN
					fbReader.eCmd := eEnumCmd_Next;
					IF ( nRow <= csv_rows ) THEN
						IF ( nColumn <= csv_columns ) THEN
							database[nRow, nColumn] := CSVFIELD_TO_STRING( sCSVField, FALSE );
						END_IF
					END_IF
				END_IF
			END_FOR
			IF fbReader.bCRLF THEN(* CRLF == TRUE => End of reacord reached *)
				nColumn := 0;
			END_IF
		END_FOR
		step := 10;

	10:	(* Close source file *)
		fbFileClose( bExecute := FALSE );
		fbFileClose( sNetId := sNetId, hFile := hFile, bExecute := TRUE );
		step := 11;

	11:(* Wait until close not busy *)
		fbFileClose( bExecute := FALSE, bError => bError, nErrID => nErrID );
		IF ( NOT fbFileClose.bBusy ) THEN
			hFile := 0;
			step := 100;
		END_IF

	100: (* Error or ready step => cleanup *)
		IF ( hFile <> 0 ) THEN
			step := 10; (* Close the source file *)
		ELSE
			bBusy := FALSE;
			error := bError;
			step := 0;	(* Ready *)
		END_IF

END_CASE

END_FUNCTION_BLOCK

// ---- POUs/Data/FB_SavePar.TcPOU
FUNCTION_BLOCK FB_SavePar
VAR_IN_OUT
	
	motorAix:FB_MotorMovements;
	saveRef:DataSaveModule_EX;
	gStaParSet:ST_StationConfigBase;
	languageswitch:BOOL;
	logOut:printLogModule_EX;
END_VAR
VAR_INPUT
	chinnesename:WSTRING;
	eglishname:	STRING;
	pos1name:WSTRING;
	bigSizeFocPosname:STRING;
	RunVelname:STRING;
	
	saveIndexOffset:INT;
END_VAR
VAR_OUTPUT
	moveerro:BOOL;
	movebusy:BOOL;
	movedone:BOOL;
END_VAR
VAR
	step:INT;
	loadTon:TON;
	loadR_Trig:R_Trig;
	saveTon:TON;
	saveR_Trig:R_Trig;
	wstrShow:WSTRING:="";
END_VAR

movedone:=FALSE;
gStaParSet.AixChineseName:=chinnesename;
gStaParSet.AixEnglishName:=eglishname;
gStaParSet.pos1name:=pos1name;
gStaParSet.movetopos1btname:="";
IF gCNErrShow THEN
	gStaParSet.movetopos1btname:=wconcat(gStaParSet.movetopos1btname,"移动到");
ELSE
	gStaParSet.movetopos1btname:=wconcat(gStaParSet.movetopos1btname,"MoveTo");
END_IF

gStaParSet.movetopos1btname:=wconcat(gStaParSet.movetopos1btname,pos1name);

gStaParSet.savepos1btname:="";
IF gCNErrShow THEN
	gStaParSet.savepos1btname:=wconcat(gStaParSet.savepos1btname,"保存");
ELSE
	gStaParSet.savepos1btname:=wconcat(gStaParSet.savepos1btname,"Save");
END_IF
gStaParSet.savepos1btname:=wconcat(gStaParSet.savepos1btname,pos1name);

gStaParSet.AixActPos:=motorAix.Get_ActPos();
gStaParSet.AixActVel:=motorAix.Get_ActVel();
IF languageswitch THEN
	gStaParSet.AixNameShow:=gStaParSet.AixChineseName;
ELSE
	gStaParSet.AixNameShow:=TO_WSTRING(gStaParSet.AixEnglishName);
END_IF
IF gStaParSet.Move_Pos1 THEN
	step:=100;
	gStaParSet.Move_Pos1:=FALSE;
END_IF

saveTon(IN:=gsave, PT:=T#2S, Q=> , ET=> );
saveR_Trig(CLK:=gsave , Q=> );
IF gStaParSet.SavePar THEN
	gStaParSet.Pos1:=motorAix.Get_ActPos();
	wstrShow:=WCONCAT(wstrShow,chinnesename);
	wstrShow:=WCONCAT(wstrShow," ");
	wstrShow:=WCONCAT(wstrShow,TO_WSTRING(gStaParSet.Pos1));
	logOut.append_EX(wstrShow);
	wstrShow:="";
	gStaParSet.SavePar:=FALSE;
END_IF
IF saveR_Trig.Q  THEN 
	saveRef.setLrealValue(gStaParSet.Pos1,1*INT_TO_UDINT(saveIndexOffset)+0);
END_IF
IF saveTon.Q THEN
	gSaveTemp:=TRUE;
	gsave:=FALSE;
END_IF


IF gRead  THEN
	saveRef.getLrealValue(gStaParSet.Pos1,1*INT_TO_UDINT(saveIndexOffset)+0);
END_IF

IF fbMachineState.Reset THEN
	step:=0;
	moveerro:=FALSE;
	gStaParSet.Reset:=FALSE;
	movebusy:=FALSE;
	motorAix.Act_RESET();
END_IF
IF gStaParSet.Stop THEN
	gStaParSet.Stop:=FALSE;
	motorAix.Act_STOP();
	step:=0;
	movebusy:=FALSE;
END_IF

CASE step OF
	0:
		;
	100:
		IF NOT motorAix.Get_Busy() AND motorAix.Get_HomeState() AND motorAix.Get_AbsCondition() THEN
			step:=110;
			movebusy:=TRUE;
			motorAix.Act_ABS(gStaParSet.Pos1,gStaParSet.RunVel);
		ELSE
			step:=300;
		END_IF
	110:
		//新增功能2
		IF motorAix.Get_Done_Abs() THEN
			step:=0;
			movebusy:=FALSE;
		END_IF
		IF motorAix.Get_Error() THEN
			step:=300;
		END_IF
		
	300:
		moveerro:=TRUE;
		step:=0;
END_CASE

END_FUNCTION_BLOCK

// ---- POUs/BaseModule/UPS_CX51X0/ups_CX51X0.TcPOU
PROGRAM ups_CX51X0
VAR_INPUT
	bWrtie					: BOOL;//触发保存
END_VAR
VAR
	//fbUPS					: FB_S_UPS;
	fbUPS					: FB_S_UPS_CX51x0;
	fbGetCurTaskIndex		: GetCurTaskIndex;
	fbWritePersistentData	: FB_WritePersistentData;
	nTaskNo					: INT;
	wrtieR_TRIG				: R_TRIG;
END_VAR

(* 需要在变量改变之后, PLC断电之前触发bWrtie *)
wrtieR_TRIG(CLK:=bWrtie);

fbGetCurTaskIndex(index=>nTaskNo);
fbWritePersistentData(
	NETID:= , 
	PORT:= 851, 
	START:= wrtieR_TRIG.Q OR TwinCAT_SystemInfoVarList._TaskInfo[nTaskNo].FirstCycle, 
	TMOUT:= , 
	MODE:= , 
	BUSY=> , 
	ERR=> , 
	ERRID=> );

IF wrtieR_TRIG.Q THEN
	bWrtie:=FALSE;
END_IF

(* 以下仅用于带1s UPS的CX51x0 PLC *)
fbUPS(
	sNetID:= , 
	iPLCPort:= 851, 
	iUPSPort:= , 
	tTimeout:= , 
	eUpsMode:= , 
	ePersistentMode:= , 
	tRecoverTime:= , 
	bPowerFailDetect=> , 
	eState=> );

METHOD Act_Wrtie
VAR_INPUT
END_VAR
bWrtie:=TRUE;
END_METHOD

ACTION VersionLog:
(*
版本: V1.0.0.0
说明:
	1. 首个版本
(**************************************************)
版本: V1.0.0.1
说明:
	1. 修正断电保持失效功能
(**************************************************)
版本: V1.0.0.2
说明:
	1. 怎么函数Act_Wrtie()，方便外部调用
(**************************************************)
*)
END_ACTION

END_PROGRAM

// ---- POUs/Other/MainRunPOU.TcPOU
PROGRAM MainRunPOU
VAR_INPUT
	HomeInit:BOOL;
	AllInit:BOOL;
	AllPause:BOOL;
	AllAbort:BOOL;
	stopToClear:BOOL;
	warningCount:BOOL;
	tempLoadNumber:UDINT;
	bigCamRatio:REAL;
	smallCamRatio:REAL;
	canModify:BOOL;
	testLog:BOOL;
END_VAR

VAR 
	DelayStart:TON;
	DelayFlag:BOOL:=TRUE;	

	autoRun_R_Trig:R_TRIG;
	autoRun_F_Trig:F_TRIG;
	autoRun_F_Trig1:F_TRIG;
	pause1_R_Trig:R_TRIG;
	pause2_R_Trig:R_TRIG;
	
	
	StartRunTon:TON;
	StartRunR:R_TRIG;
	ResetButR:R_trig;
	
	
	fAxisOverride:LREAL;
	fAxisOverride1:LREAL;
	
	quitAutoRun:BOOL:=FALSE;
	stop_F_Trig:F_Trig;
	stop_F_Trig1:F_Trig;
	itemp: INT;
	testpp:BOOL;
	stopToClearTON:TON;
	useWarningRtrig:R_TRIG;
	WarningRtrig:R_TRIG;
	fFtrigSW:F_TRIG;
	nCfgSlaveCount AT%I*:UINT;//绑定，Device 1:Input : SlaveCount
	nSlaveCount AT%I*:UINT;//绑定，Device 1:InfoData : CfgSlaveCount
	ErrorR_Trig							:R_Trig;
	ErrorF_Trig							:F_Trig;
	testTON:TON;
	notbusyTON							:TON;
	testLogRtrig:R_TRIG;
	testLogTimes:UINT:=0;
	forceEnableRecovery:TON;
END_VAR

gVersion:='V1.0.29';// 
//gPosDeviation:=0.001; // 位置偏差
	(* Other *) 
 	//Instance 对象的实例化最好先执行
//	gEnablePDVSWConnect:=TRUE;
//	gEnableSRFSWConnect:=TRUE;
//	gEnablePRFSWConnect:=TRUE;
//	gEnableHeGSWConnect:=TRUE;
 	InstanceUtility();
	//加入该延迟目的是为了使系统时钟初始化后能被正确调用。
	DelayStart(IN:=DelayFlag , PT:=T#5S , Q=> , ET=> );
	IF DelayStart.Q THEN
		DelayFlag:=FALSE;
		gRecipeNameMax:=gRecipeNameMax;
		gRead:=TRUE;//读取
		gCNErrShow:=FALSE;
	END_IF
	IF DelayFlag THEN
		RETURN;
	END_IF
	instance();//轴、气缸、电磁阀实例化
 	//MachineState机台状态刷新
	MachineStatePOU();
	otherMachineState();
	PRG_ADS_Comm_ByName_A2B();// ADS通讯刷新
	// 通讯
	FuncModule_RS232_SRF();
	FuncModule_RS232_ARM();
	FuncModule_RS485_MFC();
//	FuncModule_RS232_TBP();
//	FuncModule_RS232_ARM();
	errorMonitor();
	ACT_ErrorMonitor();
	//DownTimeRecord宕机时间记录
	DownTimeRecordPOU();
	
	ACT_LogTest();
(* 半自动动作复位、暂停处理*)
	S_CO_ControlRF(bInit:=AllInit, bPause:=AllPause, bAbort:=AllAbort);
	S_PDVSafeCtr(bInit:=AllInit, bPause:=AllPause, bAbort:=AllAbort);
	S_ActuatorRecoveryPOU(bInit:=AllInit, bPause:=AllPause, bAbort:=AllAbort);
	S_BackOfHeliumClear(bInit:=AllInit, bPause:=AllPause, bAbort:=AllAbort);
	S_RoughPumping(bInit:=AllInit, bPause:=AllPause, bAbort:=AllAbort);
	
	S_LoadLockVent(bInit:=AllInit, bPause:=AllPause, bAbort:=AllAbort);
	S_ChamberLLVent(bInit:=AllInit, bPause:=AllPause, bAbort:=AllAbort);
	S_MachineVent(bInit:=AllInit, bPause:=AllPause, bAbort:=AllAbort);
	
	S_LoadWafer(bInit:=AllInit, bPause:=AllPause, bAbort:=AllAbort);
	S_Etching(bInit:=AllInit, bPause:=AllPause, bAbort:=AllAbort);
	S_UnLoadWafer(bInit:=AllInit, bPause:=AllPause, bAbort:=AllAbort);
	
	MainPOU(bInit:=AllInit, bPause:=AllPause, bAbort:=AllAbort);
	IF HomeInit THEN
		HomeInit:=FALSE;
	END_IF
	IF AllInit THEN
		AllInit:=FALSE;
	END_IF
	IF AllAbort THEN
		AllAbort:=FALSE;
	END_IF
	IF gErrorAbort THEN
		AllAbort:=TRUE;
		HomeInit:=TRUE;
		AllInit:=TRUE;
		AllPause:=FALSE;
	END_IF
	
 (* 进入自动*)
	autoRun_R_Trig(CLK:=gAutoRunningFlag);
	IF autoRun_R_Trig.Q THEN
		HomeInit:=TRUE;
		AllInit:=TRUE;
		AllAbort:=TRUE;
		AllPause:=FALSE;
		gLog.append_EX(" 进入自动");
		gDataChangeLog.append_EX("进入自动");
		fb_systemTimeModule.startTime(14);//总时间开始计时
	END_IF
	StartRunTon(IN:=gAutoRunningFlag,PT:=T#1000MS);// 等待各个模组复位完成
	StartRunR(CLK:=StartRunTon.Q);
	IF StartRunR.Q THEN
		MainPOU.Act_init_status();
		MainPOU.Act_Ex();
		MainPOU.bTrig:=TRUE;//暂时屏蔽
	END_IF
 (* 退出自动*)
 	notbusyTON(IN:=NOT gSPOUBusy AND gCtrlMode=ControlMode.eAutoCtrMode,PT:=T#2S);
 	IF notbusyTON.Q THEN
		gAutoRunningFlag:=FALSE;
		gCtrlMode:=ControlMode.eManualCtrMode;
		HomeInit:=TRUE;
		AllInit:=TRUE;
		AllAbort:=TRUE;
		AllPause:=FALSE;
	END_IF
 	autoRun_F_Trig(CLK:=gAutoRunningFlag);
	IF autoRun_F_Trig.Q THEN		
		HomeInit:=TRUE;
		AllInit:=TRUE;
		AllAbort:=TRUE;
		AllPause:=FALSE;
		gDataChangeLog.append_EX(" 退出自动");
	END_IF
 (* 进入暂停*)
	pause1_R_Trig(CLK:=(gAutoRunningFlag AND (gRunningState=RunningStatus.eErrorState) OR (gRunningState=RunningStatus.ePauseState)));
	IF pause1_R_Trig.Q THEN
		AllPause:=TRUE;
	END_IF
 (* 退出暂停*)
	pause2_R_Trig(CLK:=(gAutoRunningFlag AND (gRunningState=RunningStatus.eAutoState)));
	IF pause2_R_Trig.Q THEN
		AllPause:=FALSE;
	END_IF
 (*复位按钮动作*)
 	ResetButR(CLK:=fbMachineState.Reset , Q=> );
	IF ResetButR.Q THEN
		;
	END_IF
IF nCfgSlaveCount<>nSlaveCount THEN//nSlaveCount在Device1的Inputs_SlaveCount中；nCfgSlaveCount在Device1中的InfoData中的CfgSlaveCount中
	error_Trigger(5);// 报警提示有从站掉线
END_IF
ErrorR_Trig(CLK:=(gRunningState=RunningStatus.eErrorState) AND (gCtrlMode=3 OR ((gRunningState<>RunningStatus.eHomeState)) AND NOT gAutoRunningFlag), Q=> );//
ErrorF_Trig(CLK:=(gRunningState=RunningStatus.eErrorState) AND (gCtrlMode=3 OR ((gRunningState<>RunningStatus.eHomeState)) AND NOT gAutoRunningFlag), Q=> );//
forceEnableRecovery(IN:=gEnablePDVOpenClose OR gEnableGDOpenClose OR gEnableHeInOpenClose,PT:=T#20S);
IF forceEnableRecovery.Q THEN
	gEnablePDVOpenClose:=FALSE;
	gEnableGDOpenClose:=FALSE;
	gEnableHeInOpenClose:=FALSE;
END_IF
//IF ErrorR_Trig.Q THEN//报错停止操作
//	AllPause:=TRUE;
//END_IF
//IF ErrorF_Trig.Q THEN
//	AllPause:=FALSE;
//END_IF

ACTION ACT_ErrorMonitor:
IF NOT gDisablePressureCheck THEN
	IF gICP.I_PressureCheck THEN
		error_Trigger(50);
	END_IF
END_IF

IF NOT gDisableWaterFloweCheck THEN
	IF gICP.I_WaterFlowCheck THEN
		error_Trigger(51);
	END_IF
END_IF

IF NOT gDisableWaterTemCheck THEN
	IF gICP.I_WaterTemperatureCheck THEN
		error_Trigger(51);
	END_IF
END_IF

IF gICP.ForeLineGauge.error THEN
	error_Trigger(53);
END_IF
IF gICP.LoadLockGauge.error THEN
	error_Trigger(54);
END_IF
IF gICP.AIMGauge.error THEN
	error_Trigger(55);
END_IF
IF gICP.ChamberGauge.error THEN
	error_Trigger(56);
END_IF
IF gICP.TBGauge.error THEN
	error_Trigger(58);
END_IF
END_ACTION

ACTION ACT_LogTest:
testLogRtrig(CLK:=testLog);
IF testLogRtrig.Q THEN
	gDataChangeLog.append(CONCAT('Pressure is:',REAL_TO_STRING(gICP.HeCheckGaugeReal)));
	gDataChangeLog.append(CONCAT('MFC flow is:',REAL_TO_STRING(gICP.HeMFC_SetFlowHMI)));
END_IF
testTON(IN:=NOT testTON.Q AND testLog, PT:= T#1S, Q=> , ET=> );
IF testTON.Q THEN
	testLogTimes:=testLogTimes+1;
	gDataChangeLog.append(CONCAT('Pressure is:',REAL_TO_STRING(gICP.HeCheckGaugeReal)));
	IF testLogTimes>=29 THEN
		testLogTimes:=0;
		testLog:=FALSE;
	END_IF
END_IF
END_ACTION

ACTION allAxisStop:
//临时使用，当做停机使用
END_ACTION

ACTION VersonRecord:
//硬件 配置更新，需更改加减速度\IO 还核定
//上料逻辑已完成，下料逻辑差POU以及Other Cal吸嘴距离的计算等内容

//1.0.0 第一次调试
//1.0.2 Recipe测试基本满足需求 20241028
//1.0.3 TB GASLINE界面、底层块操作验证
//1.0.4 除了RF、Load外，其余已经与UI同步
//1.0.5 UI除了LoadLock没操作，其余已同步完成；IO硬件绑定盒信号关联已完成
//1.0.6 RS232 通讯测试-字符串测试已完成
//1.0.7 RS232 通讯测试-RR匹配器通讯测试，当前位置匹配不正确
//1.0.8 RS232 TB只是预先编写完成，还未进行测试；  Chiller的通讯底层已经完成，还未进行验证测试
//1.0.9	Chiller的网口通讯测试完成
//1.0.10	Chiller的网口通讯测试完成;PDV测试完成，但是对于Pressure Aligment的时候，存在小数点的向上向下取整的问题；
//1.0.11	带操作提示；--下一版本需求，操作确认提示为可选项
//1.0.12	带操作提示完善；--下一版本需求，操作确认提示为可选项;
//1.0.13	GAS BOX Valve 等控件组合状态及控制
//1.0.14	操作提示、二次确认、半自动
//1.0.15	ADS通讯变量
//1.0.20    PDV、ARM、LoadLock、Valve等都已调试
//1.0.21    GAS BOX、分子泵等都已调试；测试没问题
//1.0.22   差RF的起破测试
//1.0.23   下电极RF Power正常起破::::晶圆进入腔体内记忆状态需写步骤方式完成;
//1.0.24   完善互锁（PDV的压力控制模式需要谨慎考虑，特别是没有气体进入的时候）;
//1.0.25   操作提示完善
//1.0.26   互锁条件完善
//1.0.27   互锁条件完善,POU完善
//1.0.28   互锁完善
//1.0.29   程序逻辑进一步完善
END_ACTION

END_PROGRAM

// ---- POUs/Instance/InstanceUtility.TcPOU
PROGRAM InstanceUtility
VAR
	systemTime1						: TIMESTRUCT;

END_VAR

(*********** 公共部分 ***********)
(*log对象 实例化*)

	gLog(
		sRootDirPath:= 'C:\Log', 
		sFileName:= 'All_Log.txt', 
		enable:=TRUE, 
		enableShowInfo:= TRUE, 
		clearShowInfo:= , 
		enableDelete:= TRUE, 
		storageDays:= 20, 
		busy=> , 
		error=> , 
		errID=> , 
		errTxt=> );
	gDownTimeLog(
		sRootDirPath:= 'C:\Log', 
		sFileName:= 'gDownTimeLog.txt', 
		enable:=TRUE , 
		enableShowInfo:= TRUE, 
		clearShowInfo:= , 
		enableDelete:= TRUE, 
		storageDays:= 20, 
		busy=> , 
		error=> , 
		errID=> , 
		errTxt=> );
	gDataChangeLog(
		sRootDirPath:= 'C:\Log', 
		sFileName:= 'gDataChangeLog.txt', 
		enable:= TRUE, 
		enableShowInfo:= TRUE, 
		clearShowInfo:= , 
		enableDelete:= TRUE, 
		storageDays:= 20, 
		busy=> , 
		error=> , 
		errID=> , 
		errTxt=> );
	gOperatorLog(
		sRootDirPath:= 'C:\Log', 
		sFileName:= 'gOperatorLog.txt', 
		enable:= TRUE, 
		enableShowInfo:= TRUE, 
		clearShowInfo:= , 
		enableDelete:= TRUE, 
		storageDays:= 30, 
		busy=> , 
		error=> , 
		errID=> , 
		errTxt=> );
	gRunningLog(
		sRootDirPath:= 'C:\Log', 
		sFileName:= 'gRunningLog.txt', 
		enable:= TRUE, 
		enableShowInfo:= TRUE, 
		clearShowInfo:= , 
		enableDelete:= TRUE, 
		storageDays:= 30, 
		busy=> , 
		error=> , 
		errID=> , 
		errTxt=> );
	
(*通用对象 实例化*)/////////////////////////////////////////////////////计时内容可以根据情况删减

	fb_systemTimeModule(systemTime=>systemTime1 , timeInterval=> );//时钟实例化
	g_SystemTime:=fb_systemTimeModule.getStrSysTime();//界面现实时间
	
	fb_systemTimeModule.enableTime(11);// Load cycle time 统计
	fb_systemTimeModule.enableTime(12);// Test cycle time 统计
	fb_systemTimeModule.enableTime(13);// UnLoad cycle time 统计
	fb_systemTimeModule.enableTime(14);// Toltal cycle time 统计
	fb_systemTimeModule.enableTime(15);// Test BreakDOwm cycle time 统计
	
//	fb_systemTimeModule.enableTime(20);
//	fb_systemTimeModule.enableTime(30);
//	fb_systemTimeModule.enableTime(31);
//	fb_systemTimeModule.enableTime(32);
//	// fb_systemTimeModule.enableTime(33);
//	fb_systemTimeModule.enableTime(35);
//	fb_systemTimeModule.enableTime(36);
//	fb_systemTimeModule.enableTime(37);
//	fb_systemTimeModule.enableTime(38);
//	// fb_systemTimeModule.enableTime(50);
	
//	// fb_systemTimeModule.enableTime(100);
	
//	fb_systemTimeModule.enableTime(200);
	
	

	
//	fb_systemTimeModule.enableTime(500);
//	fb_systemTimeModule.enableTime(510);
	
//// Sta1	
//	fb_systemTimeModule.enableTime(610);// Sta1 Load Time
//	fb_systemTimeModule.enableTime(611);// Sta1 Time of Load Pos to Test Start Pos
//	fb_systemTimeModule.enableTime(612);// Sta1 Time of Test End Pos to UnLoad Pos
//	fb_systemTimeModule.enableTime(613);// Sta1 TestTime
//	fb_systemTimeModule.enableTime(614);// Sta1 UnLoad Time
//	fb_systemTimeModule.enableTime(615);// Sta1 Time of UnLoad Pos to Load Pos

END_PROGRAM

// ---- POUs/Instance/instance.TcPOU
PROGRAM instance
VAR
	testbool:BOOL;
	test:struct_byte;
	
	arryRtrig:ARRAY [1..10] OF  R_TRIG;
	allMFCSetStep:UINT;
	setTon:TON;
	setTimeOut:BOOL;
	allMFCClearStep:UINT;
	clearTON:TON;
	clearTimeOut:BOOL;
	timeOutTime:TIME:=T#5S;
	setdoneRecoveryTON:TON;
	cleardoneRecoveryTON:TON;
	setEqualTON:TON;
	gvaOpenRtrig:R_TRIG;
	gvaCloseRtrig:R_TRIG;
	gvbOpenRtrig:R_TRIG;
	gvbCloseRtrig:R_TRIG;
	mfcSetRtrig:R_TRIG;
	mfcClearRtrig:R_TRIG;
	conditionTon:ARRAY [1..10] OF  TON;
	conditionTonRTrig:ARRAY [1..10] OF  R_TRIG;
	heinStep:INT:=0;
	heoutStep:INT:=0;
	heOldset:REAL;
END_VAR


	PLC_SW1.logHandleArray[1]:=ADR(gLog);
	PLC_SW1.logHandleArrayLength:=1;
	PLC_SW1(
		nSocketType:=1 , //配置Server\Client
		sTerminalName:='PLC_SW1' , 
		sHost:=gRemoteHostIp , //gRemoteHost, gLocalHost, '127.0.0.1',
		nPort:=gRemoteHostPort , 
		bEnable:=gEnableSWConnect , 
		sSendSuffix:='$R$N',
		nQueueInterval:=10 , //配置发送队列间隔时间 单位ms
		logHandleArray:= , 
		logHandleArrayLength:= , 
		bSendCondition=> , 
		bSocketConnected=>gSWConnected );
		
